// TwinCAT 3 PLC project Library
// Title: lcls-twincat-motion
// Company: SLAC
// ProjectVersion: 0.0.0
// ProgramVersion: 3.1.4026.17
// libraries:
//   LCLS General, * (SLAC)
//   lcls-twincat-math, * (SLAC - LCLS)
//   LCLS_OOPMotion, * (SLAC)
//   PMPS, * (SLAC - LCLS)
//   Tc2_EtherCAT, * (Beckhoff Automation GmbH)
//   Tc2_Math, * (Beckhoff Automation GmbH)
//   Tc2_MC2, * (Beckhoff Automation GmbH)
//   Tc2_Standard, * (Beckhoff Automation GmbH)
//   Tc2_System, * (Beckhoff Automation GmbH)
//   Tc2_Utilities, * (Beckhoff Automation GmbH)
//   Tc3_IPCDiag, * (Beckhoff Automation GmbH)
//   Tc3_JsonXml, * (Beckhoff Automation GmbH)
//   Tc3_Module, * (Beckhoff Automation GmbH)
//   TcUnit, * (www.tcunit.org)
// project tree:
//   DUTs/Deprecated/ ENUM_MotionRequest.TcDUT, DUT_MotionPneumaticActuator.TcDUT, DUT_MotionStage.TcDUT, DUT_PositionState.TcDUT, EL5042_Status.TcDUT, ENUM_EpicsHomeCmd.TcDUT, ENUM_EpicsInOut.TcDUT, ENUM_EpicsInOut_INT.TcDUT, ENUM_EpicsMotorCmd.TcDUT, ENUM_MotionFFType.TcDUT, ENUM_PnuematicActuatorPositionState.TcDUT, ENUM_StageBrakeMode.TcDUT, ENUM_StageEnableMode.TcDUT, ENUM_StatePMPSStatus.TcDUT
//   DUTs/DS402/ E_DS402DriveState.TcDUT, E_DS402EGU.TcDUT, E_MCS2HomeMethod.TcDUT, E_MCS2OpMode.TcDUT, E_MCS2OpModeReq.TcDUT, E_HomeStates.TcDUT (not stored), E_Module.TcDUT, E_MoveDoneCause.TcDUT, E_MoveMode.TcDUT, E_MoveState.TcDUT, E_StartupState.TcDUT, ST_ChannelState.TcDUT, ST_DS402Drive.TcDUT, ST_DS402DriveStatus.TcDUT (not stored), ST_MCS2ChanParameter.TcDUT
//   DUTs/ E_EpicsHomeCmd.TcDUT, ST_AxisParameterSetExposed.TcDUT, E_LCLSMotionError.TcDUT, E_MotionFFType.TcDUT, E_StatePMPSStatus.TcDUT, ST_MotionEpicsInterface.TcDUT, ST_MotionStage.TcDUT, ST_PositionState.TcDUT, ST_StateEpicsToPlc.TcDUT, ST_StatePlcToEpics.TcDUT, ST_StatePMPSEpicsToPlc.TcDUT, ST_EL5042_Status.TcDUT, E_EpicsInOut.TcDUT, E_EpicsMotorCmd.TcDUT, E_MotionRequest.TcDUT, E_StageBrakeMode.TcDUT, E_StageEnableMode.TcDUT, ST_MotionPneumaticActuator.TcDUT, E_PnuematicActuatorPositionState.TcDUT, ST_RenishawAbsEnc.TcDUT, ST_StatePMPSPlcToEpics.TcDUT
//   GVLs/ MOTION_GVL.TcGVL, MotionConstants.TcGVL
//   / PlcTask.TcTTO
//   POUs/Deprecated/ FB_EpicsInOut.TcPOU, FB_PositionStateBase.TcPOU, FB_PositionStateBase_WithPMPS.TcPOU, FB_PositionStateBase_WithPMPS_Test.TcPOU, FB_PositionStateInOut.TcPOU, FB_PositionStateInOut_WithPMPS.TcPOU, FB_PositionStateInOut_WithPMPS_Test.TcPOU, FB_PositionStateManager.TcPOU, FB_PositionStatePMPS.TcPOU, FB_PositionStatePMPS_Base.TcPOU, FB_PositionStatePMPS_Test.TcPOU, FB_StatePTPMove.TcPOU
//   POUs/ImplicitChecks/ CheckBounds.TcPOU, CheckDivDInt.TcPOU, CheckDivLInt.TcPOU, CheckDivLReal.TcPOU, CheckDivReal.TcPOU
//   POUs/Motion/DS402/ FB_MotionStageE727.TcPOU (excluded from build)
//   POUs/Motion/DS402/MCS2/ FB_MCS2Calibrate.TcPOU, FB_MCS2DriveManager.TcPOU, FB_MCS2Home.TcPOU, FB_MCS2ReadParams.TcPOU (excluded from build), FB_MCS2StepMode.TcPOU, FB_MotionStageMCS2.TcPOU, FB_ReadChanParameters.TcPOU, FB_ReadDriveCodes.TcPOU, FB_WriteCalibrationParameters.TcPOU (excluded from build), FB_WriteHomeParameters.TcPOU (excluded from build), FB_WriteChanParameters.TcPOU, F_MCS2ErrorCodeLookup.TcPOU, FB_WriteStepModeParameters.TcPOU (excluded from build)
//   POUs/Motion/ FB_EncoderValue.TcPOU, FB_EncSaveRestore.TcPOU, FB_LogMotionError.TcPOU, FB_MotionBacklashCompensation.TcPOU, FB_MotionHoming.TcPOU, FB_MotionRequest.TcPOU, FB_MotionStage.TcPOU, FB_MotionStageNCParams.TcPOU, FB_MotionStageSim.TcPOU, FB_MotionPneumaticActuator.TcPOU, FB_MotionVirtualFrame.TcPOU
//   POUs/Motion/Gantry/ FB_GantryAutoCoupling.TcPOU, FB_GantryDiffVirtualLimitSwitch.TcPOU
//   POUs/Motion/PMPS/ FB_EncErrorFFO.TcPOU, FB_MiscStatesErrorFFO.TcPOU, FB_MotionBPTM.TcPOU, FB_MotionClearAsserts.TcPOU, FB_MotionReadPMPSDBND.TcPOU, FB_PerMotorFFOND.TcPOU, FB_NCErrorFFO.TcPOU, FB_PositionStatePMPS1D.TcPOU, FB_PositionStatePMPS2D.TcPOU, FB_PositionStatePMPS3D.TcPOU, FB_PositionStatePMPSND_Core.TcPOU, FB_Standard_PMPSDB.TcPOU, FB_StatePMPSEnables.TcPOU, FB_StatePMPSEnablesND.TcPOU
//   POUs/Motion/States/Examples/ FB_PositionState1D_InOut.TcPOU, FB_PositionStatePMPS2D_InOut.TcPOU, FB_PositionStatePMPS1D_InOut.TcPOU, FB_PositionState2D_InOut.TcPOU
//   POUs/Motion/States/ FB_PositionState2D.TcPOU, FB_PositionState3D.TcPOU, FB_PositionStateND_Core.TcPOU, FB_PositionStateMove.TcPOU, FB_PositionState1D.TcPOU, FB_PositionStateMoveND.TcPOU, FB_PositionStateRead.TcPOU, FB_PositionStateReadND.TcPOU, FB_StateSetupHelper.TcPOU, FB_StatesInputHandler.TcPOU
//   POUs/Motion/States/Helpers/ FB_RawCountConverter.TcPOU, F_AtPositionState.TcPOU, F_PosOverLowerBound.TcPOU, F_PosUnderUpperBound.TcPOU, F_PosWithinDelta.TcPOU
//   POUs/Motion/States/Internals/ FB_PositionStateInternal.TcPOU, FB_PositionStateInternalND.TcPOU, FB_PositionStateLock.TcPOU
//   POUs/Motion/Utils/ FB_SetEnables.TcPOU, F_MotionErrorCodeLookup.TcPOU
//   POUs/MotorTesting/ FB_MicroStepCountTest.TcPOU
//   tc_mca_std_lib/DUTs/ DUT_AxisStatus_v0_01.TcDUT (not stored)
//   tc_mca_std_lib/GVLs/ GVL.TcGVL (not stored)
//   tc_mca_std_lib/POUs/ChangeConfig/ FB_ReadFloatParameter.TcPOU (not stored), FB_ReadParameterInNc_v1_00.TcPOU (not stored), FB_WriteFloatParameter.TcPOU (not stored), FB_WriteParameterInNc_v1_00.TcPOU (not stored)
//   tc_mca_std_lib/POUs/ErrorHandling/ DUT_ErrorState.TcDUT (not stored), DUT_TerminalError.TcDUT (not stored), FB_ErrorList.TcPOU (not stored), FB_TerminalError.TcPOU (not stored), GVL_ErrorSystem.TcGVL (not stored), ST_ErrorSystem.TcDUT (not stored)
//   tc_mca_std_lib/POUs/Hardware/EtherCAT_Terminals/Analog_Inputs/ EL3174_0002.TcPOU (not stored), EL3214.TcPOU (not stored), EL3255.TcPOU (not stored), FB_CalculateFrequency_3702_v0_01.TcPOU (not stored)
//   tc_mca_std_lib/POUs/Hardware/EtherCAT_Terminals/Digital_Inputs/ EL1008.TcPOU (not stored), EL1018.TcPOU (not stored), EL1808.TcPOU (not stored), EL1809.TcPOU (not stored), EL1819.TcPOU (not stored), FB_EL1252ASM_v1_00.TcPOU (not stored)
//   tc_mca_std_lib/POUs/Hardware/EtherCAT_Terminals/Digital_Outputs/ EL2014.TcPOU (not stored), EL2252.TcPOU (not stored), EL2808.TcPOU (not stored), EL2819.TcPOU (not stored)
//   tc_mca_std_lib/POUs/Hardware/EtherCAT_Terminals/Digital_Outputs/External_Types/ dutEL2521_Ctrl.TcDUT (not stored), dutEL2521_Status.TcDUT (not stored)
//   tc_mca_std_lib/POUs/Hardware/EtherCAT_Terminals/Measuring_Terminals/ EL5002.TcPOU (not stored), EL5021.TcPOU (not stored), EL5042.TcPOU (not stored), EL5101.TcPOU (not stored)
//   tc_mca_std_lib/POUs/Hardware/EtherCAT_Terminals/Motion/ EL7211_v1_00.TcPOU (not stored), EL9576_v1_00.TcPOU (not stored)
//   tc_mca_std_lib/POUs/Hardware/EtherCAT_Terminals/System/ EL9410.TcPOU (not stored), EL9505.TcPOU (not stored)
//   tc_mca_std_lib/POUs/Hardware/Other/ EK1200.TcPOU (not stored)
//   tc_mca_std_lib/POUs/Motion/ FB_DriveVirtual.TcPOU (not stored), FB_NcAxis.TcPOU (not stored)
//   tc_mca_std_lib/POUs/Motion/Homing/ FB_HomeDirect.TcPOU (not stored), FB_HomeFinish.TcPOU (not stored), FB_HomePrepare.TcPOU (not stored), FB_HomeReadNcVelocities.TcPOU (not stored), FB_HomeReadSoftLimEnable.TcPOU (not stored), FB_HomeToSwitch.TcPOU (not stored), FB_HomeVirtual.TcPOU (not stored), FB_HomeWriteNcVelocities.TcPOU (not stored), FB_HomeWriteSoftLimEnable.TcPOU (not stored)
//   Tests/ FB_AtPositionState_Test.TcPOU, FB_AxisParameterSetExposed_Test.TcPOU, FB_MiscStatesErrorFFO_Test.TcPOU, FB_MotionBPTM_Test.TcPOU, FB_MCS2DriveManager_Test.TcPOU, FB_MotionClearAsserts_Test.TcPOU, FB_MotionReadPMPSDBND_Test.TcPOU, FB_MotionVirtualFrame_Test.TcPOU, FB_NCErrorFFO_Test.TcPOU, FB_PerMotorFFOND_Test.TcPOU, FB_PositionStateMoveND_Test.TcPOU, FB_PositionStateMove_Test.TcPOU, FB_PositionStatePMPSND_Test.TcPOU, FB_PositionStateReadND_Test.TcPOU, FB_PositionStateRead_Test.TcPOU, FB_PositionStateND_Test.TcPOU, FB_PowerEnableMode_Test.TcPOU, FB_MotionBacklashCompensation_Test.TcPOU, FB_StatePMPSEnablesND_Test.TcPOU, FB_StatePMPSEnables_Test.TcPOU, FB_StateSetupHelper_Test.TcPOU, FB_TestHelperSetAndMove_Test.TcPOU, FB_TestStateInitTiming.TcPOU, PRG_TEST.TcPOU
//   Tests/Helpers/ E_TestStates.TcDUT, FB_CauseNCError.TcPOU, FB_MotionStageSetAndMoveHelper.TcPOU, FB_MotionStageSetHelper.TcPOU, FB_MotorTestSuite.TcPOU, FB_PMPSJsonTestHelper.TcPOU, FB_TestHelperSetAndMove.TcPOU
// real-time tasks:
//   TASK PlcTask: cycle T#10ms, priority 20, ADS port 350
// motion (NC):
//   TASK NC-Task 1 SAF: cycle T#1ms, priority 4, ADS port 501
//   TASK NC-Task 1 SVB: cycle T#10ms, priority 8, ADS port 511
//   AXIS Axis_PositionStateRead_Test (id 3)
//     OtherSettings: AllowMotionCmdToSlave=true
//     encoder EncType=1
//     drive DrvType=5
//       Analog: ScaleFactorActTorque=0.1
//     controller CtrType=1
//       CtrPara: PriorControlFactor=1
//         Observer: BandWidth=20
//   AXIS Axis_AtPositionState_Test (id 4)
//     OtherSettings: AllowMotionCmdToSlave=true
//     encoder EncType=1
//     drive DrvType=5
//       Analog: ScaleFactorActTorque=0.1
//     controller CtrType=1
//       CtrPara: PriorControlFactor=1
//         Observer: BandWidth=20
//   AXIS Axis_TestHelperSetAndMove_Test (id 5)
//     OtherSettings: AllowMotionCmdToSlave=true
//     encoder EncType=1
//     drive DrvType=5
//       Analog: ScaleFactorActTorque=0.1
//     controller CtrType=1
//       CtrPara: PriorControlFactor=1
//         Observer: BandWidth=20
//   AXIS Axis_PositionStateReadND_Test_1 (id 6)
//     OtherSettings: AllowMotionCmdToSlave=true
//     encoder EncType=1
//     drive DrvType=5
//       Analog: ScaleFactorActTorque=0.1
//       TimeComp: TaskDelayCycles=1
//     controller CtrType=1
//       CtrPara: PriorControlFactor=1
//         Observer: BandWidth=20
//   AXIS Axis_PositionStateReadND_Test_2 (id 7)
//     OtherSettings: AllowMotionCmdToSlave=true
//     encoder EncType=1
//     drive DrvType=5
//       Analog: ScaleFactorActTorque=0.1
//       TimeComp: TaskDelayCycles=1
//     controller CtrType=1
//       CtrPara: PriorControlFactor=1
//         Observer: BandWidth=20
//   AXIS Axis_PositionStateReadND_Test_3 (id 8)
//     OtherSettings: AllowMotionCmdToSlave=true
//     encoder EncType=1
//     drive DrvType=5
//       Analog: ScaleFactorActTorque=0.1
//       TimeComp: TaskDelayCycles=1
//     controller CtrType=1
//       CtrPara: PriorControlFactor=1
//         Observer: BandWidth=20
//   AXIS Axis_PositionStateMove_Test (id 9)
//     OtherSettings: AllowMotionCmdToSlave=true
//     encoder EncType=1
//     drive DrvType=5
//       Analog: ScaleFactorActTorque=0.1
//     controller CtrType=1
//       CtrPara: PriorControlFactor=1
//         Observer: BandWidth=20
//   AXIS Axis_PositionStateMoveND_Test_1 (id 10)
//     OtherSettings: AllowMotionCmdToSlave=true
//     encoder EncType=1
//     drive DrvType=5
//       Analog: ScaleFactorActTorque=0.1
//     controller CtrType=1
//       CtrPara: PriorControlFactor=1
//         Observer: BandWidth=20
//   AXIS Axis_PositionStateMoveND_Test_2 (id 11)
//     OtherSettings: AllowMotionCmdToSlave=true
//     encoder EncType=1
//     drive DrvType=5
//       Analog: ScaleFactorActTorque=0.1
//     controller CtrType=1
//       CtrPara: PriorControlFactor=1
//         Observer: BandWidth=20
//   AXIS Axis_PositionStateMoveND_Test_3 (id 12)
//     OtherSettings: AllowMotionCmdToSlave=true
//     encoder EncType=1
//     drive DrvType=5
//       Analog: ScaleFactorActTorque=0.1
//     controller CtrType=1
//       CtrPara: PriorControlFactor=1
//         Observer: BandWidth=20
//   AXIS Axis_PositionStateND_Test_1 (id 13)
//     OtherSettings: AllowMotionCmdToSlave=true
//     encoder EncType=1
//     drive DrvType=5
//       Analog: ScaleFactorActTorque=0.1
//       TimeComp: TaskDelayCycles=1
//     controller CtrType=1
//       CtrPara: PriorControlFactor=1
//         Observer: BandWidth=20
//   AXIS Axis_PositionStateND_Test_2 (id 14)
//     OtherSettings: AllowMotionCmdToSlave=true
//     encoder EncType=1
//     drive DrvType=5
//       Analog: ScaleFactorActTorque=0.1
//       TimeComp: TaskDelayCycles=1
//     controller CtrType=1
//       CtrPara: PriorControlFactor=1
//         Observer: BandWidth=20
//   AXIS Axis_PositionStateND_Test_3 (id 15)
//     OtherSettings: AllowMotionCmdToSlave=true
//     encoder EncType=1
//     drive DrvType=5
//       Analog: ScaleFactorActTorque=0.1
//       TimeComp: TaskDelayCycles=1
//     controller CtrType=1
//       CtrPara: PriorControlFactor=1
//         Observer: BandWidth=20
//   AXIS Axis_NCErrorFFO_Test (id 16)
//     OtherSettings: AllowMotionCmdToSlave=true
//     encoder EncType=1
//     drive DrvType=5
//       Analog: ScaleFactorActTorque=0.1
//     controller CtrType=1
//       CtrPara: PriorControlFactor=1
//         Observer: BandWidth=20
//   AXIS Axis_PositionStatePMPSND_Test_1 (id 17)
//     OtherSettings: AllowMotionCmdToSlave=true
//     encoder EncType=1
//     drive DrvType=5
//       Analog: ScaleFactorActTorque=0.1
//     controller CtrType=1
//       CtrPara: PriorControlFactor=1
//         Observer: BandWidth=20
//   AXIS Axis_PositionStatePMPSND_Test_2 (id 18)
//     OtherSettings: AllowMotionCmdToSlave=true
//     encoder EncType=1
//     drive DrvType=5
//       Analog: ScaleFactorActTorque=0.1
//     controller CtrType=1
//       CtrPara: PriorControlFactor=1
//         Observer: BandWidth=20
//   AXIS Axis_PositionStatePMPSND_Test_3 (id 19)
//     OtherSettings: AllowMotionCmdToSlave=true
//     encoder EncType=1
//     drive DrvType=5
//       Analog: ScaleFactorActTorque=0.1
//     controller CtrType=1
//       CtrPara: PriorControlFactor=1
//         Observer: BandWidth=20
//   AXIS Axis_StatePMPSEnable_Test (id 20)
//     OtherSettings: AllowMotionCmdToSlave=true
//     encoder EncType=1
//     drive DrvType=5
//       Analog: ScaleFactorActTorque=0.1
//       TimeComp: TaskDelayCycles=1
//     controller CtrType=1
//       CtrPara: PriorControlFactor=1
//         Observer: BandWidth=20
//   AXIS Axis_PositionStateReadND_Test_4 (id 21)
//     OtherSettings: AllowMotionCmdToSlave=true
//     encoder EncType=1
//     drive DrvType=5
//       Analog: ScaleFactorActTorque=0.1
//     controller CtrType=1
//       CtrPara: PriorControlFactor=1
//         Observer: BandWidth=20
//   AXIS Axis_PositionStateReadND_Test_5 (id 22)
//     OtherSettings: AllowMotionCmdToSlave=true
//     encoder EncType=1
//     drive DrvType=5
//       Analog: ScaleFactorActTorque=0.1
//     controller CtrType=1
//       CtrPara: PriorControlFactor=1
//         Observer: BandWidth=20
//   AXIS Axis_TestStateInitTiming (id 1)
//     OtherSettings: AllowMotionCmdToSlave=true
//     encoder EncType=1
//     drive DrvType=5
//       Analog: TorqueSetpointScale=10, ScaleFactorActTorque=0.1
//     controller CtrType=1
//       CtrPara: PriorControlFactor=1
//         Observer: BandWidth=20
//   AXIS Axis_AxisParameter_Test (id 2)
//     Dynamic: AccelerationMaximum=2, DecelerationMaximum=3
//     Velo: Maximum=1
//     PositionAreaControl: Range=1
//     OtherSettings: AllowMotionCmdToSlave=true
//     encoder EncType=1
//       EncPara: Offset=12
//         SoftEndMinControl: Enable=true, Range=4
//         SoftEndMaxControl: Enable=true, Range=5
//     drive DrvType=5
//       Analog: TorqueSetpointScale=10, ScaleFactorActTorque=0.1
//       TimeComp: TaskDelayCycles=1
//     controller CtrType=1
//       CtrPara: PriorControlFactor=1
//         PosDiffControl: Range=6, Time=7
//         Observer: BandWidth=20
//   AXIS Axis_PowerEnableMode_Test (id 29) // Test axis for stmotionStage Axis Power Enable Mode control
//     OtherSettings: AllowMotionCmdToSlave=true
//     encoder EncType=1
//     drive DrvType=5
//       Analog: TorqueSetpointScale=10, ScaleFactorActTorque=0.1
//       TimeComp: TaskDelayCycles=1
//     controller CtrType=1
//       CtrPara: PriorControlFactor=1
//         Observer: BandWidth=20
//   AXIS Axis_BacklashCompensation_Test (id 30)
//     OtherSettings: AllowMotionCmdToSlave=true
//     encoder EncType=1
//       ActPosCorrection: Enable=true
//     drive DrvType=5
//       Analog: TorqueSetpointScale=10, ScaleFactorActTorque=0.1
//     controller CtrType=1
//       CtrPara: PriorControlFactor=1
//         Observer: BandWidth=20
//   AXIS Axis_NewArchMcMotionBlocks_Test (id 31)
//     OtherSettings: AllowMotionCmdToSlave=true
//     encoder EncType=1
//     drive DrvType=5
//       Analog: TorqueSetpointScale=10, ScaleFactorActTorque=0.1
//       TimeComp: TaskDelayCycles=1
//     controller CtrType=1
//       CtrPara: PriorControlFactor=1
//         Observer: BandWidth=20
//   AXIS Axis_MotionVirtualFrameRx_Test (id 23)
//     OtherSettings: AllowMotionCmdToSlave=true
//     encoder EncType=1
//     drive DrvType=5
//       Analog: TorqueSetpointScale=10, ScaleFactorActTorque=0.1
//     controller CtrType=1
//       CtrPara: PriorControlFactor=1
//         Observer: BandWidth=20
//   AXIS Axis_MotionVirtualFrameRy_Test (id 24)
//     OtherSettings: AllowMotionCmdToSlave=true
//     encoder EncType=1
//     drive DrvType=5
//       Analog: TorqueSetpointScale=10, ScaleFactorActTorque=0.1
//     controller CtrType=1
//       CtrPara: PriorControlFactor=1
//         Observer: BandWidth=20
//   AXIS Axis_MotionVirtualFrameRz_Test (id 25)
//     OtherSettings: AllowMotionCmdToSlave=true
//     encoder EncType=1
//     drive DrvType=5
//       Analog: TorqueSetpointScale=10, ScaleFactorActTorque=0.1
//     controller CtrType=1
//       CtrPara: PriorControlFactor=1
//         Observer: BandWidth=20
//   AXIS Axis_MotionVirtualFrameVx_Test (id 26)
//     OtherSettings: AllowMotionCmdToSlave=true
//     encoder EncType=7
//       EncPara: ScaleFactorNumerator=1e-06, MaxCount=#xffffffff, ReferenceSystem=1
//     drive DrvType=5
//       Analog: TorqueSetpointScale=10, ScaleFactorActTorque=0.1
//       TimeComp: TaskDelayCycles=1
//     controller CtrType=1
//       CtrPara: PriorControlFactor=1
//         PosDiffControl: Enable=false
//         Observer: BandWidth=20
//   AXIS Axis_MotionVirtualFrameVy_Test (id 27)
//     OtherSettings: AllowMotionCmdToSlave=true
//     encoder EncType=7
//       EncPara: ScaleFactorNumerator=1e-06, MaxCount=#xffffffff, ReferenceSystem=1
//     drive DrvType=5
//       Analog: TorqueSetpointScale=10, ScaleFactorActTorque=0.1
//       TimeComp: TaskDelayCycles=1
//     controller CtrType=1
//       CtrPara: PriorControlFactor=1
//         PosDiffControl: Enable=false
//         Observer: BandWidth=20
//   AXIS Axis_MotionVirtualFrameVz_Test (id 28)
//     OtherSettings: AllowMotionCmdToSlave=true
//     encoder EncType=7
//       EncPara: ScaleFactorNumerator=1e-06, MaxCount=#xffffffff, ReferenceSystem=1
//     drive DrvType=5
//       Analog: TorqueSetpointScale=10, ScaleFactorActTorque=0.1
//       TimeComp: TaskDelayCycles=1
//     controller CtrType=1
//       CtrPara: PriorControlFactor=1
//         PosDiffControl: Enable=false
//         Observer: BandWidth=20
// variable links:
//   Library Instance <-> NC-Task 1 SAF/Axes/Axis_AtPositionState_Test
//     PlcTask Inputs/PRG_TEST.fb_AtPositionState_Test.stMotionStage.Axis.NcToPlc <-> Outputs/ToPlc
//     PlcTask Outputs/PRG_TEST.fb_AtPositionState_Test.stMotionStage.Axis.PlcToNc <-> Inputs/FromPlc
//   Library Instance <-> NC-Task 1 SAF/Axes/Axis_AxisParameter_Test
//     PlcTask Inputs/PRG_TEST.fb_AxisParameterSetExposed_Test.stMotionStage.Axis.NcToPlc <-> Outputs/ToPlc
//     PlcTask Outputs/PRG_TEST.fb_AxisParameterSetExposed_Test.stMotionStage.Axis.PlcToNc <-> Inputs/FromPlc
//   Library Instance <-> NC-Task 1 SAF/Axes/Axis_BacklashCompensation_Test
//     PlcTask Inputs/PRG_TEST.fb_MotionBacklashCompensation_Test.stMotionStage.Axis.NcToPlc <-> Outputs/ToPlc
//     PlcTask Outputs/PRG_TEST.fb_MotionBacklashCompensation_Test.stMotionStage.Axis.PlcToNc <-> Inputs/FromPlc
//   Library Instance <-> NC-Task 1 SAF/Axes/Axis_MotionVirtualFrameRx_Test
//     PlcTask Inputs/PRG_TEST.fbMotionVirtualFrameTest.stMotionStageRx.Axis.NcToPlc <-> Outputs/ToPlc
//     PlcTask Outputs/PRG_TEST.fbMotionVirtualFrameTest.stMotionStageRx.Axis.PlcToNc <-> Inputs/FromPlc
//   Library Instance <-> NC-Task 1 SAF/Axes/Axis_MotionVirtualFrameRy_Test
//     PlcTask Inputs/PRG_TEST.fbMotionVirtualFrameTest.stMotionStageRy.Axis.NcToPlc <-> Outputs/ToPlc
//     PlcTask Outputs/PRG_TEST.fbMotionVirtualFrameTest.stMotionStageRy.Axis.PlcToNc <-> Inputs/FromPlc
//   Library Instance <-> NC-Task 1 SAF/Axes/Axis_MotionVirtualFrameRz_Test
//     PlcTask Inputs/PRG_TEST.fbMotionVirtualFrameTest.stMotionStageRz.Axis.NcToPlc <-> Outputs/ToPlc
//     PlcTask Outputs/PRG_TEST.fbMotionVirtualFrameTest.stMotionStageRz.Axis.PlcToNc <-> Inputs/FromPlc
//   Library Instance <-> NC-Task 1 SAF/Axes/Axis_MotionVirtualFrameVx_Test
//     PlcTask Inputs/PRG_TEST.fbMotionVirtualFrameTest.stMotionStageVx.Axis.NcToPlc <-> Outputs/ToPlc
//     PlcTask Outputs/PRG_TEST.fbMotionVirtualFrameTest.nPositionCountsVx <-> Enc/Inputs/In/nDataIn1
//     PlcTask Outputs/PRG_TEST.fbMotionVirtualFrameTest.stMotionStageVx.Axis.PlcToNc <-> Inputs/FromPlc
//   Library Instance <-> NC-Task 1 SAF/Axes/Axis_MotionVirtualFrameVy_Test
//     PlcTask Inputs/PRG_TEST.fbMotionVirtualFrameTest.stMotionStageVy.Axis.NcToPlc <-> Outputs/ToPlc
//     PlcTask Outputs/PRG_TEST.fbMotionVirtualFrameTest.nPositionCountsVy <-> Enc/Inputs/In/nDataIn1
//     PlcTask Outputs/PRG_TEST.fbMotionVirtualFrameTest.stMotionStageVy.Axis.PlcToNc <-> Inputs/FromPlc
//   Library Instance <-> NC-Task 1 SAF/Axes/Axis_MotionVirtualFrameVz_Test
//     PlcTask Inputs/PRG_TEST.fbMotionVirtualFrameTest.stMotionStageVz.Axis.NcToPlc <-> Outputs/ToPlc
//     PlcTask Outputs/PRG_TEST.fbMotionVirtualFrameTest.nPositionCountsVz <-> Enc/Inputs/In/nDataIn1
//     PlcTask Outputs/PRG_TEST.fbMotionVirtualFrameTest.stMotionStageVz.Axis.PlcToNc <-> Inputs/FromPlc
//   Library Instance <-> NC-Task 1 SAF/Axes/Axis_NCErrorFFO_Test
//     PlcTask Inputs/PRG_TEST.fb_NCErrorFFO_Test.stMotionStage.Axis.NcToPlc <-> Outputs/ToPlc
//     PlcTask Outputs/PRG_TEST.fb_NCErrorFFO_Test.stMotionStage.Axis.PlcToNc <-> Inputs/FromPlc
//   Library Instance <-> NC-Task 1 SAF/Axes/Axis_PositionStateMoveND_Test_1
//     PlcTask Inputs/PRG_TEST.fb_PositionStateMoveND_Test.astMotionStage[1].Axis.NcToPlc <-> Outputs/ToPlc
//     PlcTask Outputs/PRG_TEST.fb_PositionStateMoveND_Test.astMotionStage[1].Axis.PlcToNc <-> Inputs/FromPlc
//   Library Instance <-> NC-Task 1 SAF/Axes/Axis_PositionStateMoveND_Test_2
//     PlcTask Inputs/PRG_TEST.fb_PositionStateMoveND_Test.astMotionStage[2].Axis.NcToPlc <-> Outputs/ToPlc
//     PlcTask Outputs/PRG_TEST.fb_PositionStateMoveND_Test.astMotionStage[2].Axis.PlcToNc <-> Inputs/FromPlc
//   Library Instance <-> NC-Task 1 SAF/Axes/Axis_PositionStateMoveND_Test_3
//     PlcTask Inputs/PRG_TEST.fb_PositionStateMoveND_Test.astMotionStage[3].Axis.NcToPlc <-> Outputs/ToPlc
//     PlcTask Outputs/PRG_TEST.fb_PositionStateMoveND_Test.astMotionStage[3].Axis.PlcToNc <-> Inputs/FromPlc
//   Library Instance <-> NC-Task 1 SAF/Axes/Axis_PositionStateMove_Test
//     PlcTask Inputs/PRG_TEST.fb_PositionStateMove_Test.stMotionStage.Axis.NcToPlc <-> Outputs/ToPlc
//     PlcTask Outputs/PRG_TEST.fb_PositionStateMove_Test.stMotionStage.Axis.PlcToNc <-> Inputs/FromPlc
//   Library Instance <-> NC-Task 1 SAF/Axes/Axis_PositionStateND_Test_1
//     PlcTask Inputs/PRG_TEST.fb_PositionStateND_Test.stMotionStage1.Axis.NcToPlc <-> Outputs/ToPlc
//     PlcTask Outputs/PRG_TEST.fb_PositionStateND_Test.stMotionStage1.Axis.PlcToNc <-> Inputs/FromPlc
//   Library Instance <-> NC-Task 1 SAF/Axes/Axis_PositionStateND_Test_2
//     PlcTask Inputs/PRG_TEST.fb_PositionStateND_Test.stMotionStage2.Axis.NcToPlc <-> Outputs/ToPlc
//     PlcTask Outputs/PRG_TEST.fb_PositionStateND_Test.stMotionStage2.Axis.PlcToNc <-> Inputs/FromPlc
//   Library Instance <-> NC-Task 1 SAF/Axes/Axis_PositionStateND_Test_3
//     PlcTask Inputs/PRG_TEST.fb_PositionStateND_Test.stMotionStage3.Axis.NcToPlc <-> Outputs/ToPlc
//     PlcTask Outputs/PRG_TEST.fb_PositionStateND_Test.stMotionStage3.Axis.PlcToNc <-> Inputs/FromPlc
//   Library Instance <-> NC-Task 1 SAF/Axes/Axis_PositionStatePMPSND_Test_1
//     PlcTask Inputs/PRG_TEST.fb_PositionStatePMPSND_Test.stMotionStage1.Axis.NcToPlc <-> Outputs/ToPlc
//     PlcTask Outputs/PRG_TEST.fb_PositionStatePMPSND_Test.stMotionStage1.Axis.PlcToNc <-> Inputs/FromPlc
//   Library Instance <-> NC-Task 1 SAF/Axes/Axis_PositionStatePMPSND_Test_2
//     PlcTask Inputs/PRG_TEST.fb_PositionStatePMPSND_Test.stMotionStage2.Axis.NcToPlc <-> Outputs/ToPlc
//     PlcTask Outputs/PRG_TEST.fb_PositionStatePMPSND_Test.stMotionStage2.Axis.PlcToNc <-> Inputs/FromPlc
//   Library Instance <-> NC-Task 1 SAF/Axes/Axis_PositionStatePMPSND_Test_3
//     PlcTask Inputs/PRG_TEST.fb_PositionStatePMPSND_Test.stMotionStage3.Axis.NcToPlc <-> Outputs/ToPlc
//     PlcTask Outputs/PRG_TEST.fb_PositionStatePMPSND_Test.stMotionStage3.Axis.PlcToNc <-> Inputs/FromPlc
//   Library Instance <-> NC-Task 1 SAF/Axes/Axis_PositionStateReadND_Test_1
//     PlcTask Inputs/PRG_TEST.fb_PositionStateReadND_Test.astMotionStage[1].Axis.NcToPlc <-> Outputs/ToPlc
//     PlcTask Outputs/PRG_TEST.fb_PositionStateReadND_Test.astMotionStage[1].Axis.PlcToNc <-> Inputs/FromPlc
//   Library Instance <-> NC-Task 1 SAF/Axes/Axis_PositionStateReadND_Test_2
//     PlcTask Inputs/PRG_TEST.fb_PositionStateReadND_Test.astMotionStage[2].Axis.NcToPlc <-> Outputs/ToPlc
//     PlcTask Outputs/PRG_TEST.fb_PositionStateReadND_Test.astMotionStage[2].Axis.PlcToNc <-> Inputs/FromPlc
//   Library Instance <-> NC-Task 1 SAF/Axes/Axis_PositionStateReadND_Test_3
//     PlcTask Inputs/PRG_TEST.fb_PositionStateReadND_Test.astMotionStage[3].Axis.NcToPlc <-> Outputs/ToPlc
//     PlcTask Outputs/PRG_TEST.fb_PositionStateReadND_Test.astMotionStage[3].Axis.PlcToNc <-> Inputs/FromPlc
//   Library Instance <-> NC-Task 1 SAF/Axes/Axis_PositionStateReadND_Test_4
//     PlcTask Inputs/PRG_TEST.fb_PositionStateReadND_Test.astSqMotionStage[1].Axis.NcToPlc <-> Outputs/ToPlc
//     PlcTask Outputs/PRG_TEST.fb_PositionStateReadND_Test.astSqMotionStage[1].Axis.PlcToNc <-> Inputs/FromPlc
//   Library Instance <-> NC-Task 1 SAF/Axes/Axis_PositionStateReadND_Test_5
//     PlcTask Inputs/PRG_TEST.fb_PositionStateReadND_Test.astSqMotionStage[2].Axis.NcToPlc <-> Outputs/ToPlc
//     PlcTask Outputs/PRG_TEST.fb_PositionStateReadND_Test.astSqMotionStage[2].Axis.PlcToNc <-> Inputs/FromPlc
//   Library Instance <-> NC-Task 1 SAF/Axes/Axis_PositionStateRead_Test
//     PlcTask Inputs/PRG_TEST.fb_PositionStateRead_Test.stMotionStage.Axis.NcToPlc <-> Outputs/ToPlc
//     PlcTask Outputs/PRG_TEST.fb_PositionStateRead_Test.stMotionStage.Axis.PlcToNc <-> Inputs/FromPlc
//   Library Instance <-> NC-Task 1 SAF/Axes/Axis_PowerEnableMode_Test
//     PlcTask Inputs/PRG_TEST.fb_PowerEnableMode_Test.stMotionStage.Axis.NcToPlc <-> Outputs/ToPlc
//     PlcTask Outputs/PRG_TEST.fb_PowerEnableMode_Test.stMotionStage.Axis.PlcToNc <-> Inputs/FromPlc
//   Library Instance <-> NC-Task 1 SAF/Axes/Axis_StatePMPSEnable_Test
//     PlcTask Inputs/PRG_TEST.fb_StatePMPSEnables_Test.stMotionStage.Axis.NcToPlc <-> Outputs/ToPlc
//     PlcTask Outputs/PRG_TEST.fb_StatePMPSEnables_Test.stMotionStage.Axis.PlcToNc <-> Inputs/FromPlc
//   Library Instance <-> NC-Task 1 SAF/Axes/Axis_TestHelperSetAndMove_Test
//     PlcTask Inputs/PRG_TEST.fb_TestHelperSetAndMove_Test.stMotionStage.Axis.NcToPlc <-> Outputs/ToPlc
//     PlcTask Outputs/PRG_TEST.fb_TestHelperSetAndMove_Test.stMotionStage.Axis.PlcToNc <-> Inputs/FromPlc
//   Library Instance <-> NC-Task 1 SAF/Axes/Axis_TestStateInitTiming
//     PlcTask Inputs/PRG_TEST.fb_TestStateInitTiming.stMotionStage.Axis.NcToPlc <-> Outputs/ToPlc
//     PlcTask Outputs/PRG_TEST.fb_TestStateInitTiming.stMotionStage.Axis.PlcToNc <-> Inputs/FromPlc

CONFIGURATION Library
    RESOURCE PLC ON TwinCAT3
        TASK PlcTask(INTERVAL := T#10ms, PRIORITY := 20);
        PROGRAM PRG_TEST WITH PlcTask : PRG_TEST;
    END_RESOURCE
END_CONFIGURATION

// ---- DUTs/Deprecated/ENUM_MotionRequest.TcDUT
{attribute 'obsolete' := 'Use E_MotionRequest'}
TYPE ENUM_MotionRequest : E_MotionRequest; END_TYPE

// ---- DUTs/Deprecated/DUT_MotionPneumaticActuator.TcDUT
{attribute 'obsolete' := 'DUT_MotionPneumaticActuator has been renamed to ST_MotionPneumaticActuator'}
TYPE DUT_MotionPneumaticActuator : ST_MotionPneumaticActuator; END_TYPE

// ---- DUTs/Deprecated/DUT_MotionStage.TcDUT
{attribute 'obsolete' := 'DUT_MotionStage has been renamed to ST_MotionStage'}
TYPE DUT_MotionStage : ST_MotionStage; END_TYPE

// ---- DUTs/Deprecated/DUT_PositionState.TcDUT
{attribute 'obsolete' := 'DUT_PositionState has been renamed to ST_PositionState'}
TYPE DUT_PositionState : ST_PositionState; END_TYPE

// ---- DUTs/Deprecated/EL5042_Status.TcDUT
{attribute 'obsolete' := 'EL5042_Status has been renamed to ST_EL5042_Status'}
TYPE EL5042_Status : ST_EL5042_Status; END_TYPE

// ---- DUTs/Deprecated/ENUM_EpicsHomeCmd.TcDUT
{attribute 'obsolete' := 'Use E_EpicsHomeCmd'}
TYPE ENUM_EpicsHomeCmd : E_EpicsHomeCmd; END_TYPE

// ---- DUTs/Deprecated/ENUM_EpicsInOut.TcDUT
{attribute 'obsolete' := 'Use E_EpicsInOut'}
TYPE ENUM_EpicsInOut : E_EpicsInOut; END_TYPE

// ---- DUTs/Deprecated/ENUM_EpicsInOut_INT.TcDUT
{attribute 'obsolete' := 'Use ENUM_EpicsInOut'}
{attribute 'qualified_only'}
// Example EPICS states enum for use in all versions of the states FBs
// Remove strict attribute for easier handling
TYPE ENUM_EpicsInOut_INT :
(
    UNKNOWN := 0, // UNKNOWN must be in slot 0 or the FB breaks
    OUT := 1, // OUT at slot 1 is a convention
    IN := 2
) INT;
END_TYPE

// ---- DUTs/Deprecated/ENUM_EpicsMotorCmd.TcDUT
{attribute 'obsolete' := 'Use E_EpicsMotorCmd'}
TYPE ENUM_EpicsMotorCmd : E_EpicsMotorCmd; END_TYPE

// ---- DUTs/Deprecated/ENUM_MotionFFType.TcDUT
{attribute 'obsolete' := 'Use E_MotionFFType'}
TYPE ENUM_MotionFFType : E_MotionFFType; END_TYPE

// ---- DUTs/Deprecated/ENUM_PnuematicActuatorPositionState.TcDUT
{attribute 'obsolete' := 'Use E_PnuematicActuatorPositionState'}
TYPE ENUM_PnuematicActuatorPositionState : E_PnuematicActuatorPositionState; END_TYPE

// ---- DUTs/Deprecated/ENUM_StageBrakeMode.TcDUT
{attribute 'obsolete' := 'Use E_StageBrakeMode'}
TYPE ENUM_StageBrakeMode : E_StageBrakeMode; END_TYPE

// ---- DUTs/Deprecated/ENUM_StageEnableMode.TcDUT
{attribute 'obsolete' := 'Use E_StageEnableMode'}
TYPE ENUM_StageEnableMode : E_StageEnableMode; END_TYPE

// ---- DUTs/Deprecated/ENUM_StatePMPSStatus.TcDUT
{attribute 'obsolete' := 'Use E_StatePMPSStatus'}
TYPE ENUM_StatePMPSStatus : E_StatePMPSStatus; END_TYPE

// ---- DUTs/DS402/E_DS402DriveState.TcDUT
{attribute 'qualified_only'}
{attribute 'strict'}
{attribute 'to_string'}
TYPE E_DS402DriveState :
(
    INIT:=0,
    NO_FAULT:=1,
    SWITCH_ON_READY:=2,
    SWITCH_ON:=3,
    OPERATION_ENABLED:=4,
    FAULT:=5,
    FAULT_ACTIVE:=6,
    QUICK_STOP_ACTIVE:=7,
    SWITCH_ON_DISABLED:=8,
    MODE_ERROR:=9,
    WAIT	:= 10,
    DONE:=11
) UINT;
END_TYPE

// ---- DUTs/DS402/E_DS402EGU.TcDUT
{attribute 'qualified_only'}
{attribute 'strict'}
{attribute 'to_string'}
TYPE E_DS402EGU  :
(
    MM:=0,
    UM:=1,
    NM:=2
);
END_TYPE

// ---- DUTs/DS402/E_MCS2HomeMethod.TcDUT
{attribute 'qualified_only'}
{attribute 'strict'}
{attribute 'to_string'}
TYPE E_MCS2HomeMethod :
(
    AutoMethod := -1,
    CurrentPositionMethod := 37
)SINT;
END_TYPE

// ---- DUTs/DS402/E_MCS2OpMode.TcDUT
{attribute 'qualified_only'}
{attribute 'strict'}
{attribute 'to_string'}
TYPE E_MCS2OpMode :
(
    NONE := 0,
    // P-T-P target profil
    PROFILE_POSITION:=1,
    PROFIL_VELOCITY :=3,
    HOME:=6,
    // Cyclic synchronous modes
    CSP :=8,
    CSV :=9,
    CST := 10,
    CSTCA := 11,
    // smartAct MCS2 open loop
    CALIBRATE :=-1,
    STEP :=-4
) SINT;
END_TYPE

// ---- DUTs/DS402/E_MCS2OpModeReq.TcDUT
(*
    User-facing request for the MCS2 drive operating mode, exposed as an EPICS PV.
    This is the source of truth for which DS402 mode the drive runs in; the
    FB_MCS2DriveManager maps each value onto the corresponding E_DS402OpMode and
    switches the drive immediately when this value changes.
    CLOSED_LOOP (default) is closed-loop (CSP / NC) absolute motion.
*)
{attribute 'qualified_only'}
{attribute 'strict'}
{attribute 'to_string'}
TYPE E_MCS2OpModeReq :
(
    CLOSED_LOOP := 0,
    STEP := 1,
    HOME := 2,
    CALIBRATION := 3
) SINT;
END_TYPE

// ---- DUTs/DS402/E_Module.TcDUT
{attribute 'qualified_only'}
{attribute 'to_string'}
// Default CHAN 1, add 0x800 next channel
TYPE E_Module :
(
    CHAN1	:= 1,
    CHAN2	:= 2,
    CHAN3	:= 3
) WORD;
END_TYPE

// ---- DUTs/DS402/E_MoveDoneCause.TcDUT
{attribute 'qualified_only'}
{attribute 'strict'}
{attribute 'to_string'}
TYPE E_MoveDoneCause :
(
    UNKNOWN := 0,           // DEFAULT/UNCATEGORIZED
    MOVEDONE,               // ABSOLUTE MOVE COMPLETED
    STEPMOVEDONE,           // STEP/JOG MOVE COMPLETED
    HOMEDONE,               // HOMING COMPLETED
    CALIBRATIONDONE,        // CALIBRATION COMPLETED
    RESETDONE,              // RESET COMMAND COMPLETED
    HALTDONE,               // MANUAL HALT COMPLETED
    ABORTEDHOME,            // HOME ABORTED
    ABORTEDSTEPMOVE,        // STEP MOVE ABORTED
    ABORTEDCALIBRATION,     // CALIBRATION ABORTED
    REFERENCED,             // AXIS BECAME REFERENCED
    CALIBRATED              // AXIS BECAME CALIBRATED
);
END_TYPE

// ---- DUTs/DS402/E_MoveMode.TcDUT
{attribute 'qualified_only'}
{attribute 'strict'}
{attribute 'to_string'}
TYPE E_MoveMode  :
(
    DISCRETE_JOG:=0,
    DISCRETE_VELOCITY:=1,
    DISCRETE_RELATIVE:=2,
    DISCRETE_ABSOLUTE:=3,
    DISCRETE_MODULO:=4,
    DISCRETE_HOMING:=10
)INT;
END_TYPE

// ---- DUTs/DS402/E_MoveState.TcDUT
{attribute 'qualified_only'}
{attribute 'strict'}
{attribute 'to_string'}
TYPE E_MoveState :
(
    IDLING:=0,
    INIT:=10,
    STARTED:=20,
    IN_PROGRESS :=30,
    REACHED:=40,
    INTERRUPTED:=50,
    DONE:=60,
    ERROR:=-99
);
END_TYPE

// ---- DUTs/DS402/E_StartupState.TcDUT
{attribute 'qualified_only'}
{attribute 'strict'}
{attribute 'to_string'}
TYPE E_StartupState :
(
    STARTUP_IDLE:=0,
    STARTUP_CLEAR,
    STARTUP_RESET_FAULT,
    STARTUP_SHUTDOWN,
    STARTUP_SWITCH_ON,
    STARTUP_ENABLE_OP
);
END_TYPE

// ---- DUTs/DS402/ST_ChannelState.TcDUT
TYPE ST_ChannelState :
STRUCT
    {attribute 'pytmc' := '
        pv: STATE
        io: i
        field: DESC Channel state raw
    '}
    nChannelStateRaw  : DWORD;

    {attribute 'pytmc' := '
        pv: MOVING
        io: i
        field: DESC Actively moving
    '}
    bActivelyMoving         : BOOL;
    {attribute 'pytmc' := '
        pv: CLOSED_LOOP
        io: i
        field: DESC Closed loop active
    '}
    bClosedLoopActive       : BOOL;
    {attribute 'pytmc' := '
        pv: CALIBRATING
        io: i
        field: DESC Calibrating
    '}
    bCalibrating            : BOOL;
    {attribute 'pytmc' := '
        pv: REFERENCING
        io: i
        field: DESC Referencing
    '}
    bReferencing            : BOOL;
    {attribute 'pytmc' := '
        pv: MOVE_DELAYED
        io: i
        field: DESC Move delayed
    '}
    bMoveDelayed            : BOOL;
    {attribute 'pytmc' := '
        pv: SENSOR_PRESENT
        io: i
        field: DESC Sensor present
    '}
    bSensorPresent          : BOOL;
    {attribute 'pytmc' := '
        pv: CALIBRATED
        io: i
        field: DESC Is calibrated
    '}
    bIsCalibrated           : BOOL;
    {attribute 'pytmc' := '
        pv: REFERENCED
        io: i
        field: DESC Is referenced
    '}
    bIsReferenced           : BOOL;
    {attribute 'pytmc' := '
        pv: END_STOP
        io: i
        field: DESC End stop reached
    '}
    bEndStopReached         : BOOL;
    {attribute 'pytmc' := '
        pv: RANGE_LIMIT
        io: i
        field: DESC Range limit reached
    '}
    bRangeLimitReached      : BOOL;
    {attribute 'pytmc' := '
        pv: FOLLOWING_LIMIT
        io: i
        field: DESC Following limit reached
    '}
    bFollowingLimitReached  : BOOL;
    {attribute 'pytmc' := '
        pv: MOVE_FAILED
        io: i
        field: DESC Movement failed
    '}
    bMovementFailed         : BOOL;
    {attribute 'pytmc' := '
        pv: STREAMING
        io: i
        field: DESC Is streaming
    '}
    bIsStreaming            : BOOL;
    {attribute 'pytmc' := '
        pv: OVERLOAD
        io: i
        field: DESC Positioner overload
    '}
    bPositionerOverload     : BOOL;
    {attribute 'pytmc' := '
        pv: OVER_TEMP
        io: i
        field: DESC Over temperature
    '}
    bOverTemperature        : BOOL;
    {attribute 'pytmc' := '
        pv: REF_MARK
        io: i
        field: DESC Reference mark
    '}
    bReferenceMark          : BOOL;
    {attribute 'pytmc' := '
        pv: PHASED
        io: i
        field: DESC Is phased
    '}
    bIsPhased               : BOOL;
    {attribute 'pytmc' := '
        pv: FAULT
        io: i
        field: DESC Positioner fault
    '}
    bPositionerFault        : BOOL;
    {attribute 'pytmc' := '
        pv: AMP_ENABLED
        io: i
        field: DESC Amplifier enabled
    '}
    bAmplifierEnabled       : BOOL;
    {attribute 'pytmc' := '
        pv: IN_POSITION
        io: i
        field: DESC In position
    '}
    bInPosition             : BOOL;
    {attribute 'pytmc' := '
        pv: BRAKE_ENABLED
        io: i
        field: DESC Brake enabled
    '}
    bBrakeEnabled           : BOOL;
END_STRUCT
END_TYPE

// ---- DUTs/DS402/ST_DS402Drive.TcDUT
TYPE ST_DS402Drive:
STRUCT
    (* Global variables for the TPDO data from the drive. Each one is linked to the respective TPDO channel. *)
    stDriveStatus 			AT %I*	: 	ST_DS402DriveStatus;
    {attribute 'pytmc' := '
        pv: eOpModeDisplay
        io: i
        field: DESC MCS2 current operating mode
    '}
    nModeOfOperationDisplay AT %I*	: 	SINT;
    //nActualPosition 		AT %I*	: 	DINT;
    (*CSP drive mode*)
    nFollowingError 		AT %I*	: 	DINT;
    (* Global variables for the RPDO data to the drive. Each one is linked to the respective RPDO channel. *)
    // connected to I/O Task 'Control Word'
    nDriveControl			AT %Q*	:	UINT;
    // Connected to NC task Ctrl 1 and Ctrl 2
    nDriveControlNC			AT %I*	:	UINT;
    nTargetPosition 		AT %Q* 	: 	DINT;
    nModeOfOperation 		AT %Q* 	: 	SINT;
    nModeOfOperationNC 		AT %I* 	: 	SINT;
    (* Global variables for the RPDO data to the drive. Each one is linked to the respective RPDO channel. *)
    nProfilVelocity 		AT %Q* 	: 	DINT;
    nProfilAcceleration		AT %Q* 	: 	DINT;
    nProfilDecceleration	AT %Q* 	: 	DINT;
    nVelocityActualValue	AT %Q* 	: 	DINT;
    (* Global variables for the TPDO data from the drive. Each one is linked to the respective TPDO channel. *)
    nScantargetPosition		AT %Q*	: 	DINT;
    uScantargetVelocity		AT %Q*	: 	ULINT;
    (* Port Number of EtherCAT Slave *)
    nSlaveAddr	AT %I*  : UINT;
    (* EtherCAT slave ESM state, linked to the slave's InfoData.State.
       Low nibble is the state: 1=INIT, 2=PREOP, 4=SAFEOP, 8=OP. *)
    nEcatState	AT %I*  : UINT;
END_STRUCT
END_TYPE

// ---- DUTs/DS402/ST_MCS2ChanParameter.TcDUT
TYPE ST_MCS2ChanParameter :
STRUCT
    {attribute 'pytmc' := '
        pv: STEP_COUNT
        io: io
        field: DESC Open Loop Step Count
    '}
    nChanStep	: DINT := 500;

    {attribute 'pytmc' := '
        pv: STEP_EGU
        io: io
        field: DESC Step scale factor
    '}
    nChanStepEgu	: LREAL := 827.15;

    {attribute 'pytmc' := '
        pv: STEP_FREQ
        io: io
        field: DESC Step Frequency
    '}
    nChanStepFreq	: UINT := 500;

    {attribute 'pytmc' := '
        pv: STEP_VOLTAGE
        io: io
        field: DESC Step Amplitude
    '}
    nChanStepAmp	: UINT := 50;

    {attribute 'pytmc' := '
        pv: HOLD_TIME
        io: io
        field: DESC Close loop hold time
    '}
    nHoldTime	: UDINT := 30000;

    {attribute 'pytmc' := '
        pv: STEP_MOVE
        io: io
        field: ZNAM DISABLE
        field: ONAM ENABLE
        field: DESC Used to disable close loop mode
    '}
    bStepMoveCmd	: BOOL;

    {attribute 'pytmc' := '
        pv: STEP_FORWARD
        io: io
        field: DESC Jog one step count forward
    '}
    bStepForwardCmd	: BOOL;

    {attribute 'pytmc' := '
        pv: STEP_REVERSE
        io: io
        field: DESC Jog one step count backward
    '}
    bStepReverseCmd	: BOOL;

    {attribute 'pytmc' := '
        pv: MAX_CLF
        io: io
        field: DESC Max Close Loop Freq
    '}
    nMaxCloseLoopFreq     : UDINT;

    {attribute 'pytmc' := '
        pv: PTYPE
        io: io
        field: DESC Positioner Type
    '}
    nPositionerType	: UDINT;

    // Writable command pushed to 0x2004; the reader reads the drive value back
    // into it, so io:io serves both command and read-back on one symbol.
    {attribute 'pytmc' := '
        pv: CAL_OPT
        io: io
        field: DESC Calibration Options
    '}
    nCalibrationOpt       : DWORD;

    {attribute 'pytmc' := '
        pv: SENSOR_MODE
        io: io
        field: DESC Sensor Power Mode
    '}
    nSensorPowerMode      : UDINT;

    // Writable command pushed to 0x200B; the reader reads the drive value back
    // into it, so io:io serves both command and read-back on one symbol.
    {attribute 'pytmc' := '
        pv: REF_OPT
        io: io
        field: DESC Referencing Options
    '}
    nReferencingOpt       	   : DWORD;

    {attribute 'pytmc' := '
        pv: REF_TYPE
        io: i
        field: DESC Reference Type
    '}
    nReferenceType 	: UDINT;

    {attribute 'pytmc' := '
        pv: SAFE_DIR
        io: io
        field: ZNAM FORWARD
        field: ONAM BACKWARD
        field: DESC Safe direction (0x200C), Pre-Op
    '}
    nSafeDir	: BOOL;

    {attribute 'pytmc' := '
        pv: MOTOR_LOAD
        io: i
        field: DESC Motor Load
    '}
    nMotorLoad	: USINT;

    {attribute 'pytmc' := '
        pv: CHAN_TYPE
        io: io
        field: DESC Channel Type
    '}
    nChannelType          : UDINT;

    {attribute 'pytmc' := '
        pv: LSCO
        io: io
        field: DESC Logical Scale Offset
    '}
    nLogicalScaleOffset   : UDINT; // should LINT

    {attribute 'pytmc' := '
        pv: LSCI
        io: io
        field: DESC Logical Scale Inversion
    '}
    nLogicalScaleInv  	 : BOOL;

    {attribute 'pytmc' := '
        pv: DO_CALIB
        io: io
        field: DESC Calibrate command
    '}
    bCalibrationCmd : BOOL;

    // Desired drive operating mode (source of truth). Default is closed-loop (CSP) absolute motion.
    {attribute 'pytmc' := '
        pv: OPMODE_REQ
        io: o
        field: DESC DS402 op mode request (closed loop)
    '}
    eOpModeReq : E_MCS2OpModeReq := E_MCS2OpModeReq.CLOSED_LOOP;

    {attribute 'pytmc' := '
        pv: chanState
        io: i
        field: DESC Channel configuration parameters.
    '}
    stChannelState        : ST_ChannelState;

    {attribute 'pytmc' := '
        pv: HOME_MODE
        io: i
        field: DESC Vendor Homing Modes.
    '}
    eHomeMode			  : E_MCS2HomeMethod := E_MCS2HomeMethod.AutoMethod;

    {attribute 'pytmc' := '
        pv: CHANTEMP
        io: i
        field: DESC Channel Temperature
    '}
    nChannelTemp          : INT;

    {attribute 'pytmc' := '
        pv: MOVE_TYPE
        io: i
        field: DESC Movement Type
    '}
    nMovementType         : UDINT;

    {attribute 'pytmc' := '
        pv: BASE_UNIT
        io: i
        field: DESC Base Unit
    '}
    nBaseUnit             : UDINT;

    {attribute 'pytmc' := '
        pv: BASE_RES
        io: i
        field: DESC Base Resolution
    '}
    nBaseResolution       : DINT;

    {attribute 'pytmc' := '
        pv: DCIN
        io: io
        field: DESC Distance Code Inverted
    '}
    nDistCodeInv          : BOOL;

    {attribute 'pytmc' := '
        pv: POS_CTRL_OPT
        io: io
        field: DESC Positioner Control Options
    '}
    nPositionerCtrlOpt    : DWORD;

    {attribute 'pytmc' := '
        pv: ACT_MODE
        io: io
        field: DESC Actuator Mode
    '}
    nActuatorMode         : UDINT;

    {attribute 'pytmc' := '
        pv: MOTOR_LOAD_PROT
        io: io
        field: DESC Motor Load Protection Threshold
    '}
    nMotorLoadProt        : USINT;

    {attribute 'pytmc' := '
        pv: DIAG_CLF_MAX
        io: i
        field: DESC Diagnostic Closed Loop Frequency (max)
    '}
    nDiagClfMax           : UDINT;

    {attribute 'pytmc' := '
        pv: DIAG_CLF_AVG
        io: i
        field: DESC Diagnostic Closed Loop Frequency (avg)
    '}
    nDiagClfAvg           : UDINT;

    {attribute 'pytmc' := '
        pv: MCS2_ERR
        io: i
        field: DESC Last MCS2 drive error code (0x603F)
    '}
    nMCS2ErrorCode        : UINT;

    {attribute 'pytmc' := '
        pv: MCS2_ERR_MSG
        io: i
        field: DESC Decoded MCS2 drive error
    '}
    sMCS2ErrorMessage     : STRING;

    // Read-only decode of the drive's actual Referencing Options (REF_OPT,
    // 0x200B) into individual flags for verification. Command via REF_OPT.
    {attribute 'pytmc' := '
        pv: REF_OPT:START_DIR_BACK
        io: i
        field: DESC Ref start direction backward (bit0)
    '}
    bRefStartDirBackward  : BOOL;
    {attribute 'pytmc' := '
        pv: REF_OPT:REVERSE_DIR
        io: i
        field: DESC Ref reverse dir, multi-mark (bit1)
    '}
    bRefReverseDir        : BOOL;
    {attribute 'pytmc' := '
        pv: REF_OPT:AUTO_ZERO
        io: i
        field: DESC Ref auto-zero on reference found (bit2)
    '}
    bRefAutoZero          : BOOL;
    {attribute 'pytmc' := '
        pv: REF_OPT:ABORT_ENDSTOP
        io: i
        field: DESC Ref abort on end stop (bit3)
    '}
    bRefAbortOnEndStop    : BOOL;
    {attribute 'pytmc' := '
        pv: REF_OPT:CONT_ON_REF
        io: i
        field: DESC Ref continue on reference found (bit4)
    '}
    bRefContinueOnRefFound: BOOL;
    {attribute 'pytmc' := '
        pv: REF_OPT:STOP_ON_REF
        io: i
        field: DESC Ref stop on reference found (bit5)
    '}
    bRefStopOnRefFound    : BOOL;
    {attribute 'pytmc' := '
        pv: REF_OPT:INVALIDATE
        io: i
        field: DESC Ref invalidate is-ref flag (bit24)
    '}
    bRefInvalidate        : BOOL;

    // Read-only decode of the drive's actual Calibration Options (CAL_OPT,
    // 0x2004) into individual flags for verification. Command via CAL_OPT.
    {attribute 'pytmc' := '
        pv: CAL_OPT:DIR_BACK
        io: i
        field: DESC Calib move direction backward (bit0)
    '}
    bCalDirBackward       : BOOL;
    {attribute 'pytmc' := '
        pv: CAL_OPT:DETECT_DCI
        io: i
        field: DESC Calib detect dist code inv (bit1)
    '}
    bCalDetectDistCodeInv : BOOL;
    {attribute 'pytmc' := '
        pv: CAL_OPT:ADV_SENSOR
        io: i
        field: DESC Calib advanced sensor correction (bit2)
    '}
    bCalAdvSensorCorr     : BOOL;
    {attribute 'pytmc' := '
        pv: CAL_OPT:LIM_TRAVEL
        io: i
        field: DESC Calib limited travel, endstop (bit8)
    '}
    bCalLimitedTravelRange: BOOL;

    {attribute 'hide'}
    nHomeVeloFast         : UDINT;
    {attribute 'hide'}
    nSoftLimMin           : LINT;
    {attribute 'hide'}
    nSoftLimMax           : LINT;
    {attribute 'hide'}
    nHomeVeloSlow         : UDINT;
    {attribute 'hide'}
    nHomeAcc              : UDINT;
    {attribute 'hide'}
    nScaledFErrWin        : DINT;
    {attribute 'hide'}
    nHomeOffset           : DINT;
    {attribute 'hide'}
    nHomeMethod           : SINT;
    {attribute 'hide'}
    fScalingFactor		  : LREAL := 0.000001;
    {attribute 'hide'}
    fHomeAcc			  : LREAL := 0.8;
    // ====== Channel-specific object indices ======
    nSubIndex                : BYTE := 0;        // Main subindex (which channel)
    {attribute 'hide'}
    nChanFErrWinIdx          : WORD;
    {attribute 'hide'}
    nChanMotorLoadIdx        : WORD;
    {attribute 'hide'}
    nChanErrorCodeIdx        : WORD;
    {attribute 'hide'}
    nChanStepIdx             : WORD;
    {attribute 'hide'}
    nChanStepFreqIdx         : WORD;
    {attribute 'hide'}
    nChanStepAmpIdx          : WORD;
    {attribute 'hide'}
    nChanSoftLimitIdx        : WORD;
    {attribute 'hide'}
    nChanHomeOffsIdx         : WORD;
    {attribute 'hide'}
    nChanHomeMethodIdx       : WORD;
    {attribute 'hide'}
    nChanHomeVeloIdx         : WORD;
    {attribute 'hide'}
    nChanhomeAccIdx          : WORD;
    {attribute 'hide'}
    nCHanMaxCloseLoopFreqIdx : WORD;
    {attribute 'hide'}
    nChanPositionerTypeIdx   : WORD;
    {attribute 'hide'}
    nChanCalibrationOptIdx   : WORD;
    {attribute 'hide'}
    nChanSensorPowerModeIdx  : WORD;
    {attribute 'hide'}
    nChanReferencingOptIdx   : WORD;
    {attribute 'hide'}
    nChanReferenceTypeIdx    : WORD;
    {attribute 'hide'}
    nChanSafeDirIdx          : WORD;
    {attribute 'hide'}
    nChannelTypeIdx          : WORD;
    {attribute 'hide'}
    nChanStateIdx            : WORD;
    {attribute 'hide'}
    nChanLogicalScaleOfsIdx  : WORD;
    {attribute 'hide'}
    nChanLogicalScaleInvIdx  : WORD;
    {attribute 'hide'}
    nChanChannelTempIdx      : WORD;
    {attribute 'hide'}
    nChanMovementTypeIdx     : WORD;
    {attribute 'hide'}
    nChanBaseUnitIdx         : WORD;
    {attribute 'hide'}
    nChanBaseResolutionIdx   : WORD;
    {attribute 'hide'}
    nChanDistCodeInvIdx      : WORD;
    {attribute 'hide'}
    nChanPositionerCtrlOptIdx: WORD;
    {attribute 'hide'}
    nChanActuatorModeIdx     : WORD;
    {attribute 'hide'}
    nChanMotorLoadProtIdx    : WORD;
    {attribute 'hide'}
    nChanDiagClfIdx          : WORD;
    fPosition : LREAL;
    bStageReady : BOOL;
    // Temporary workaround: Avoid declaring mc_power externally from FB_MotionStage
    bOverrideDirEnable : BOOL := TRUE;
    bEnableHardwareOps : BOOL := TRUE;
    nReadTime : TIME := T#5S;
END_STRUCT
END_TYPE

// ---- DUTs/E_EpicsHomeCmd.TcDUT
{attribute 'qualified_only'}
{attribute 'strict'}
TYPE E_EpicsHomeCmd :
    // Defines the valid options for homing in FB_MotionStage
(
    LOW_LIMIT := 1, // Low limit switch
    HIGH_LIMIT := 2, // High limit switch
    HOME_VIA_LOW := 3, // Home switch via low switch
    HOME_VIA_HIGH := 4, // Home switch via high switch
    ABSOLUTE_SET := 15, // Set here to be fHomePosition
    // MCS2
    AutoMethod := -1, // DS402 Auto method; referencing routine set by positioner type
    CURRENT_POSITION_METHOD := 37,
    NONE := -99 // Do not home, ever
) := NONE;
END_TYPE

// ---- DUTs/ST_AxisParameterSetExposed.TcDUT
TYPE ST_AxisParameterSetExposed :
    // Collects the axis parameters that are intentionally exposed to EPICS.
STRUCT
    // Maximum Dynamics
    {attribute 'pytmc' := '
        pv: MaxVel
        io: i
        field: DESC Maximum commandable speed of the axis in EU/s.
    '}
    fVeloMaximum                : LREAL; // Maximum commandable speed of the axis in EU/s.
    {attribute 'pytmc' := '
        pv: MaxAccel
        io: i
        field: DESC Maximum rate of increase in speed of the axis in EU/s^2.
    '}
    fAccelerationMax            : LREAL; // Maximum rate of increase in speed of the axis in EU/s^2.
    {attribute 'pytmc' := '
        pv: MaxDecel
        io: i
        field: DESC Maximum rate of decrease in speed of the axis in EU/s^2.
    '}
    fDecelerationMax            : LREAL; // Maximum rate of decrease in speed of the axis in EU/s^2.

    // Monitoring
    {attribute 'pytmc' := '
        pv: PosLagEn
        io: i
        field: DESC TRUE if position lag monitor (also known as stall monitor) is enabled.
    '}
    bCtrlEnablePosDiffControl   : WORD;  // Enable/Disable state of Position Lag Monitor.
    {attribute 'pytmc' := '
        pv: PosLagVal
        io: i
        field: DESC Maximum magnitude of position lag in EU.
    '}
    fCtrlPosDiffMax             : LREAL; // Maximum magnitude of position lag in EU.
    {attribute 'pytmc' := '
        pv: PosLagTime
        io: i
        field: DESC Maximum allowable duration outside of maximum position lag value in seconds.
    '}
    fCtrlPosDiffMaxTime         : LREAL; // Maximum allowable duration outside of maximum position lag value in seconds.

    // Limit Switches
    {attribute 'pytmc' := '
        pv: SLimMinEn
        io: i
        field: DESC TRUE if controller static minimum limit is enabled.
    '}
    bEncEnableSoftEndMinControl : WORD;  // Enable/Disable state of controller static minimum limit.
    {attribute 'pytmc' := '
        pv: SLimMaxEn
        io: i
        field: DESC TRUE if controller static maximum limit is enabled.
    '}
    bEncEnableSoftEndMaxControl : WORD;  // Enable/Disable state of controller static maximum limit.
    {attribute 'pytmc' := '
        pv: SLimMin
        io: i
        field: DESC Minimum commandable position of the axis in EU.
    '}
    fEncSoftEndMin              : LREAL; // Minimum commandable position of the axis in EU.
    {attribute 'pytmc' := '
        pv: SLimMax
        io: i
        field: DESC Maximum commandable position of the axis in EU.
    '}
    fEncSoftEndMax              : LREAL; // Maximum commandable position of the axis in EU.

    // Encoder Evaluation
    {attribute 'pytmc' := '
        pv: EncScaling
        io: i
        field: DESC Encoder scaling numerator / denominator in EU/COUNT.
    '}
    fEncScaleFactorInternal      : LREAL; // Encoder scaling numerator / denominator in EU/COUNT.
    {attribute 'pytmc' := '
        pv: EncOffset
        io: i
        field: DESC Encoder offset in EU.
    '}
    fEncOffset                   : LREAL; // Encoder offset in EU.

END_STRUCT
END_TYPE

// ---- DUTs/E_LCLSMotionError.TcDUT
{attribute 'qualified_only'}
{attribute 'strict'}
TYPE E_LCLSMotionError :
(
    ABORTED := 16#7900,
    UNSAFE := 16#7901,
    INVALID := 16#7902,
    MCS2_FAULT := 16#7903,
    TEST := 16#FFFF
) UDINT;
END_TYPE

// ---- DUTs/E_MotionFFType.TcDUT
{attribute 'qualified_only'}
TYPE E_MotionFFType :
(
    STOPPER_FAULT := 16#1000,
    ZERO_RATE := 16#1001,
    BPTM_TIMEOUT := 16#1002,
    BPTM_ERROR := 16#1003,
    MAINT_MODE := 16#1004,
    NOT_A_STATE := 16#1005,
    INVALID_GOAL := 16#1006,
    TOO_MANY_TRIPS := 16#1007,
    BP_MISMATCH := 16#1008,
    INTERNAL_ERROR := 16#1009,
    PNEUMATIC_MOVE := 16#1010,
    MOT_GENERIC := 16#1011,
    LOW_RESERVED_NC := 16#2000,
    HIGH_RESERVED_NC := 16#20FF,
    DEVICE_MOVE := 16#2100
) UINT := MOT_GENERIC;
END_TYPE

// ---- DUTs/E_StatePMPSStatus.TcDUT
{attribute 'qualified_only'}
{attribute 'strict'}
TYPE E_StatePMPSStatus :
(
    // No other enum state describes it
    UNKNOWN := 0,
    // Moving toward a known state
    TRANSITION := 1,
    // Within a known state, not trying to leave
    AT_STATE := 2,
    // PMPS is in some way disabled, either with maint mode or arbiter disable
    DISABLED := 3
);
END_TYPE

// ---- DUTs/ST_MotionEpicsInterface.TcDUT
TYPE ST_MotionEpicsInterface :
    // Defines the EPICS interface to moving a motor in TwinCAT
STRUCT
 // Name to use for log messages, fast faults, etc.
    sName: STRING;
    // Set to gantry difference tolerance
    nGantryTol: LINT:=0;
    // Encoder count at which this axis is aligned with other axis
    nEncRef: ULINT:=0;

    (* Commands *)
    // Used internally to request enables
    bEnable: BOOL;

    // Used internally to reset errors and other state
    {attribute 'pytmc' := '
        pv: PLC:bReset
        io: io
        field: ZNAM FALSE
        field: ONAM TRUE
        field: DESC Used internally to reset errors
    '}
    bReset: BOOL;
    // Used internally and by the IOC to start or stop a move
    bExecute: BOOL;

    (* Command Args *)
    // Used internally and by the IOC to pick what kind of move to do
    nCommand: INT;
    // Used internally and by the IOC to pass additional data to some commands
    nCmdData: INT;
    // Used internally and by the IOC to pick a destination for the move
    fPosition: LREAL;
    // Used internally and by the IOC to pick a move velocity
    fVelocity: LREAL;
    // Used internally and by the IOC to pick a move acceleration
    fAcceleration: LREAL;
    // Used internally and by the IOC to pick a move deceleration
    fDeceleration: LREAL;
    // Used internally and by the IOC to pick a home position
    {attribute 'pytmc' := '
        pv: PLC:fHomePosition
        io: io
        field: DESC Used internally and by the IOC to pick home position
    '}
    fHomePosition: LREAL;

    (* Info *)
    // Unique ID assigned to each axis in the NC
    nMotionAxisID: UDINT:=0;
    (* Returns *)
    // TRUE if in the middle of a command
    bBusy: BOOL;
    // TRUE if we've done a command and it has finished
    bDone: BOOL;
    // TRUE if the motor has been homed, or does not need to be homed
    bHomed: BOOL;

    // TRUE if we're in an error state
    {attribute 'pytmc' := '
        pv: PLC:bError
        io: i
        field: ZNAM FALSE
        field: ONAM TRUE
        field: DESC TRUE if we are in an error state
        update: 100Hz notify
    '}
    bError: BOOL;
    // Error code if nonzero
    {attribute 'pytmc' := '
        pv: PLC:nErrorId
        io: i
        field: DESC Error code if nonzero
        update: 100Hz notify
    '}
    nErrorId: UDINT;
    // Message to identify the error state
    {attribute 'pytmc' := '
        pv: PLC:sErrorMessage
        io: i
        field: DESC Message to identify the error state
        update: 100Hz notify
    '}
    sErrorMessage: STRING;

    // Misc axis status information for the IOC
    stAxisStatus: tc2_mc2.ST_AxisStatus;
END_STRUCT
END_TYPE

// ---- DUTs/ST_MotionStage.TcDUT
TYPE ST_MotionStage :
    // Defines the EPICS interface to moving a motor in TwinCAT
STRUCT
    (* Hardware *)

    // PLC Axis Reference
    Axis: AXIS_REF;
    // NC Forward Limit Switch: TRUE if ok to move
    bLimitForwardEnable AT %I*: BOOL;
    // NC Backward Limit Switch: TRUE if ok to move
    bLimitBackwardEnable AT %I*: BOOL;
    // NO Home Switch: TRUE if at home
    bHome AT %I*: BOOL;
    // NC Brake Output: TRUE to release brake
    bBrakeRelease AT %Q*: BOOL;
    // NC STO Input: TRUE if ok to move
    {attribute 'pytmc' := '
        pv: PLC:bHardwareEnable
        io: i
        field: ZNAM FALSE
        field: ONAM TRUE
        field: DESC TRUE if STO not hit
    '}
    bHardwareEnable AT %I*: BOOL;

    // Raw encoder IO for ULINT (Biss-C)
    nRawEncoderULINT AT %I*: ULINT;
    // Raw encoder IO for UINT (Relative Encoders)
    nRawEncoderUINT AT %I*: UINT;
    // Raw encoder IO for INT (LVDT)
    nRawEncoderINT AT %I*: INT;
    // Raw encoder IO for INT (EL5072 LVDT)
    nRawEncoderDINT AT %I*: DINT;

    (* Psuedo-hardware *)

    // Forward enable EPS summary
    bAllForwardEnable: BOOL:=FALSE;
    // Backward enable EPS summary
    bAllBackwardEnable: BOOL:=FALSE;
    // Enable EPS summary encapsulating emergency stop button and any additional motion preventive hardware
    bAllEnable: BOOL:=FALSE;
    // Forward virtual gantry limit switch
    bGantryForwardEnable: BOOL:=FALSE;
    // Backward virtual gantry limit switch
    bGantryBackwardEnable: BOOL:=FALSE;
    // Encoder count summary, if linked above
    {attribute 'pytmc' := '
        pv: PLC:nEncoderCount
        io: i
        field: DESC Count from encoder hardware
    '}
    nEncoderCount: UDINT;
    // Forward Enable EPS struct
    {attribute 'pytmc' := '
        pv: PLC:stEPSF
        io: i
        field: DESC Forward Enable Interlocks
    '}
    stEPSForwardEnable: DUT_EPS;
    // Backward Enable EPS struct
    {attribute 'pytmc' := '
        pv: PLC:stEPSB
        io: i
        field: DESC Backward Enable Interlocks
    '}
    stEPSBackwardEnable: DUT_EPS;
    // Power Enable EPS struct
    {attribute 'pytmc' := '
        pv: PLC:stEPSP
        io: i
        field: DESC Power Interlocks
    '}
    stEPSPowerEnable: DUT_EPS;

    (* Settings *)
    // Name to use for log messages, fast faults, etc.
    sName: STRING;
    // If TRUE, we want to enable the motor independently of PMPS or other safety systems.
    bPowerSelf: BOOL:=FALSE;
    // Determines when we automatically enable the motor
    nEnableMode: E_StageEnableMode:=E_StageEnableMode.DURING_MOTION;
    // Determines when we automatically disengage the brake
    nBrakeMode: E_StageBrakeMode:=E_StageBrakeMode.IF_ENABLED;
    // Determines our encoder homing strategy
    nHomingMode: E_EpicsHomeCmd:=E_EpicsHomeCmd.NONE;
    // Set true to activate gantry EPS
    bGantryAxis: BOOL:=FALSE;

    // Set to gantry difference tolerance
    nGantryTol: LINT:=0;

    // Encoder count at which this axis is aligned with other axis
    nEncRef: ULINT:=0;

    (* Commands *)
    // Used internally to request enables
    bEnable: BOOL;
    // Used internally to reset errors and other state
    {attribute 'pytmc' := '
        pv: PLC:bReset
        io: io
        field: ZNAM FALSE
        field: ONAM TRUE
        field: DESC Used internally to reset errors
    '}
    bReset: BOOL;
    // Used internally and by the IOC to start or stop a move
    bExecute: BOOL;
    // Used by the IOC to disable an axis
    {attribute 'pytmc' := '
        pv: PLC:bUserEnable
        io: io
        field: ZNAM DISABLE
        field: ONAM ENABLE
        field: DESC Used to disable power entirely for an axis
        autosave_pass1: VAL
    '}
    bUserEnable: BOOL := 1;

    (* Shortcut Commands *)
    // Start a move to fPosition with fVelocity
    bMoveCmd: BOOL;
    // Start the homing routine
    {attribute 'pytmc' := '
        pv: PLC:bHomeCmd
        io: io
        field: DESC Start the homing routine
    '}
    bHomeCmd: BOOL;

    (* Command Args *)
    // Used internally and by the IOC to pick what kind of move to do
    nCommand: INT;
    // Used internally and by the IOC to pass additional data to some commands
    nCmdData: INT;
    // Used internally and by the IOC to pick a destination for the move
    fPosition: LREAL;
    // Used internally and by the IOC to pick a move velocity
    fVelocity: LREAL;
    // Used internally and by the IOC to pick a move acceleration
    fAcceleration: LREAL;
    // Used internally and by the IOC to pick a move deceleration
    fDeceleration: LREAL;
    // Used internally and by the IOC to pick a home position
    {attribute 'pytmc' := '
        pv: PLC:fHomePosition
        io: io
        field: DESC Used internally and by the IOC to pick home position
        autosave_pass1: VAL
    '}
    fHomePosition: LREAL;

    (* Info *)
    // Unique ID assigned to each axis in the NC
    nMotionAxisID: UDINT:=0;

    (* Returns *)
    // TRUE if done enabling
    bEnableDone: BOOL;
    // TRUE if in the middle of a command
    bBusy: BOOL;
    // TRUE if we've done a command and it has finished
    bDone: BOOL;
    // TRUE if the motor has been homed, or does not need to be homed
    bHomed: BOOL;
    // TRUE if we have safety permission to move
    bSafetyReady: BOOL;
    // TRUE if we're in an error state
    {attribute 'pytmc' := '
        pv: PLC:bError
        io: i
        field: ZNAM FALSE
        field: ONAM TRUE
        field: DESC TRUE if we are in an error state
    '}
    bError: BOOL;
    // Error code if nonzero
    {attribute 'pytmc' := '
        pv: PLC:nErrorId
        io: i
        field: DESC Error code if nonzero
    '}
    nErrorId: UDINT;
    // Message to identify the error state
    {attribute 'pytmc' := '
        pv: PLC:sErrorMessage
        io: i
        field: DESC Message to identify the error state
    '}
    sErrorMessage: STRING;
    // Internal hook for custom error messages
    sCustomErrorMessage: STRING;
    // MC_ReadParameterSet Output
    stAxisParameters: ST_AxisParameterSet;
    // NC parameters that are exposed with pytmc pragmas
    {attribute 'pytmc' := '
        pv: PLC:AxisPar
        io: i
        field: DESC Axis configuration parameters in the numerical controller.
    '}
    stAxisParametersExposed: ST_AxisParameterSetExposed;
    // True if we've updated stAxisParameters at least once
    bAxisParamsInit: BOOL;

    // Misc axis status information for the IOC
    stAxisStatus: DUT_AxisStatus_v0_01;

    (* Other status information for users of the IOC *)
    // Position lag difference
    {attribute 'pytmc' := '
        pv: PLC:fPosDiff
        io: i
        field: DESC Position lag difference
    '}
    fPosDiff: LREAL;

    (* Backlash compensation*)
    // Enabled axis backlash compensation
    {attribute 'pytmc' := '
        pv: PLC:bBacklashEn
        io: io
        field: ZNAM FALSE
        field: ONAM TRUE
        field: DESC Enable Backlash compensation
        autosave_pass1: VAL
    '}
    bUserBacklashEn: BOOL;

    // backlash compensation status
    {attribute 'pytmc' := '
        pv: PLC:bBacklasStatus
        io: i
        field: ZNAM DISABLED
        field: ONAM ENABLED
        field: DESC Backlash compensation status
    '}
    bBacklashStatus: BOOL;

    // Backlash compensation value
    {attribute 'pytmc' := '
        pv: PLC:fBacklash
        io: io
        field: DESC Backlash compensation
        autosave_pass1: VAL
    '}
    fBacklash: LREAL;

    // Current Backlash compensation value ?
    {attribute 'pytmc' := '
        pv: PLC:fCurrentBacklash
        io: i
        field: DESC Currently applied compensation
    '}
    fCurrentBacklash: LREAL;

    bRestoreDone : BOOL;
END_STRUCT
END_TYPE

// ---- DUTs/ST_PositionState.TcDUT
TYPE ST_PositionState :
    // Defines settings and current safety status for moves to specific positions for an axis
STRUCT
    // Name as queried via the NAME PV in EPICS
    {attribute 'pytmc' := '
        pv: NAME
        io: input
        field: DESC Name of this position state
    '}
    sName: STRING := 'Invalid';

    // Position associated with this state
    {attribute 'pytmc' := '
        pv: SETPOINT
        io: io
        field: DESC Axis position associated with this state
    '}
    fPosition: LREAL;

    {attribute 'pytmc' := '
        pv: ENCODER
        io: i
        field: DESC Encoder count associated with this state
    '}
    nEncoderCount: UDINT;

    // Maximum allowable deviation from fPosition while at the state
    fDelta: LREAL;

    // Speed at which to move to this state
    {attribute 'pytmc' := '
        pv: VELO
        io: io
        field: DESC Speed at which to move to this state
    '}
    fVelocity: LREAL;

    // (optional) Acceleration to use for moves to this state
    fAccel: LREAL;

    // (optional) Deceleration to use for moves to this state
    fDecel: LREAL;

    // Safety parameter. This must be set to TRUE by the PLC program to allow moves to this state. This is expected to change as conditions change.
    {attribute 'pytmc' := '
        pv: MOVE_OK
        io: i
        field: ZNAM FALSE
        field: ONAM TRUE
        field: DESC TRUE if the move would be safe
    '}
    bMoveOk: BOOL;

    // Signifies to FB_PositionStateLock that this state should be immutable
    bLocked: BOOL;

    // Set this to TRUE when you make your state. This defaults to FALSE so that uninitialized states can never be moved to
    bValid: BOOL;

    // Set this to TRUE when you want to use the raw encoder counts to define the state
    bUseRawCounts: BOOL;

    // Is set to TRUE by FB_PositionStateInternal when called
    bUpdated: BOOL;

    // We give this a state name and it is used to load parameters from the pmps database.
    stPMPS: ST_DbStateParams;
	
	// Set this to TRUE to enable use of the iSequence value to sequence moves that incorporate this state.
    {attribute 'pytmc' := '
        pv: SEQUENCE_MOVES
        io: i
        field: DESC TRUE if this state represents a state intended to be moved in sequence with other axes
    '}
	bSequenceMoves: BOOl;
	
	// Set this value to the sequence number that you want this state to have relative to other axes.
	// E.g. if this state has iSequence = 2 and it is being moved with a state with iSequence = 1, then
	// the iSequence = 1 state will be moved first and this state will only be moved after.
    {attribute 'pytmc' := '
        pv: SEQUENCE_ORDER
        io: i
        field: DESC Relative sequence order for the axis movement corresponding to this state.
    '}
	iSequenceOrder: UINT := 1;
END_STRUCT
END_TYPE

// ---- DUTs/ST_StateEpicsToPlc.TcDUT
TYPE ST_StateEpicsToPlc :
(*
    This data structure contains the standard EPICS input connection points for the state movers.

    The data in this struct flows from EPICS to the PLC.

    It includes everything except the SET PV, which cannot be included here
    as it is sourced from enum values unique to the application, and the PMPS PVs, which are
    gathered in their own data type, ST_StatePMPSEpicsToPlc. That actually means that this only
    holds the RESET PV, for now.

    nSetValue here is actively used by state blocks even though it is not exposed
    directly to EPICS. You should avoid manually modifying it or else
    you may interfere with normal operations of the state function blocks.

    For including your own ENUM input, you should pytmc pragma the PV name to end in "SET",
    and match the prefix of this FB's "RESET" PV. Then, you can include your enum
    as the eEnumSet IN_OUT var and let the EPICS IOC handle it.
*)
STRUCT
    // For internal use only. This holds new goal positions as an integer, else it is 0 if there is no new state move request. It is written to from the user's input enum.
    nSetValue: UINT;

    // Set this to TRUE to acknowledge and clear an error.
    {attribute 'pytmc' := '
        pv: RESET
        io: io
        field: ZNAM False
        field: ONAM True
    '}
    bReset: BOOL;
END_STRUCT
END_TYPE

// ---- DUTs/ST_StatePlcToEpics.TcDUT
TYPE ST_StatePlcToEpics :
(*
    This data structure contains the standard EPICS connection points for the state movers.

    The data in this struct flows from the PLC to EPICS.

    It includes everything except the GET PV, which cannot be included here
    as it is sourced from enum values unique to the application, and the PMPS PVs, which are
    gathered in their own data type, ST_StatePMPSPlcToEpics.

    nGetValue here is actively used by state blocks even though it is not exposed directly
    to EPICS. It is safe to read this value, but you should avoid modifying it, which may
    interfere with normal operations of the state function blocks.

    For including your own ENUM input, you should pytmc pragma the PV name to end in "GET",
    and match the prefix of this FB's "DONE" PV. Then, you can include your enum
    as the eEnumGet IN_OUT var and let the EPICS IOC handle it.
*)
STRUCT
    // For internal use only. This holds the current position index as an integer, else it is 0 if we are changing states or not at any particular state.
    nGetValue: UINT;
    // This will be TRUE when we are in an active state move and FALSE otherwise.
    {attribute 'pytmc' := '
        pv: BUSY
        io: i
        field: ZNAM False
        field: ONAM True
    '}
    bBusy: BOOL;
    // This will be TRUE after a move completes and FALSE otherwise.
    {attribute 'pytmc' := '
        pv: DONE
        io: i
        field: ZNAM False
        field: ONAM True
    '}
    bDone: BOOL;
    // This will be TRUE if the most recent move had an error and FALSE otherwise.
    {attribute 'pytmc' := '
        pv: ERR
        io: i
        field: ZNAM False
        field: ONAM True
    '}
    bError: BOOL;
    // This will be set to an NC error code during an error if one exists or left at 0 otherwise.
    {attribute 'pytmc' := '
        pv: ERRID
        io: i
    '}
    nErrorID: UDINT;
    // This will be set to an appropriate error message during an error if one exists or left as an empty string otherwise.
    {attribute 'pytmc' := '
        pv: ERRMSG
        io: i
    '}
    sErrorMsg: STRING;
END_STRUCT
END_TYPE

// ---- DUTs/ST_StatePMPSEpicsToPlc.TcDUT
TYPE ST_StatePMPSEpicsToPlc :
(*
    This data structure contains the standard PMPS EPICS connection points for the state movers.

    The data in this struct flows from EPICS to the PLC.
*)
STRUCT
    // User setting: TRUE to enable the arbiter, FALSE to disable it.
    {attribute 'pytmc' := '
        pv: PMPS:ARB:ENABLE
        io: io
    '}
    bArbiterEnabled: BOOL := TRUE;
    // User setting: TRUE to enable maintenance mode (Fast fault, free motion), FALSE to disable it.
    {attribute 'pytmc' := '
        pv: PMPS:MAINT
        io: io
    '}
    bMaintMode: BOOL;
END_STRUCT
END_TYPE

// ---- DUTs/ST_EL5042_Status.TcDUT
TYPE ST_EL5042_Status :
STRUCT
END_STRUCT
END_TYPE

// ---- DUTs/E_EpicsInOut.TcDUT
{attribute 'qualified_only'}
// Example EPICS states enum for use in all versions of the states FBs
// Remove strict attribute for easier handling
TYPE E_EpicsInOut :
(
    UNKNOWN := 0, // UNKNOWN must be in slot 0 or the FB breaks
    OUT := 1, // OUT at slot 1 is a convention
    IN := 2
) UINT;
END_TYPE

// ---- DUTs/E_EpicsMotorCmd.TcDUT
{attribute 'qualified_only'}
{attribute 'strict'}
TYPE E_EpicsMotorCmd :
    // Defines valid EPICS commands for nCommand
(
    JOG := 0,
    MOVE_VELOCITY := 1,
    MOVE_RELATIVE := 2,
    MOVE_ABSOLUTE := 3,
    MOVE_MODULO := 4,
    HOME := 10,
    GEAR := 30,
    CALIBRATE:=40
);
END_TYPE

// ---- DUTs/E_MotionRequest.TcDUT
{attribute 'qualified_only'}
{attribute 'strict'}
TYPE E_MotionRequest :
    // Defines behavior options for when FB_MotionRequest is run during an active move from another source
(
    WAIT := 0,
    INTERRUPT := 1,
    ABORT := 2
);
END_TYPE

// ---- DUTs/E_StageBrakeMode.TcDUT
{attribute 'qualified_only'}
{attribute 'strict'}
TYPE E_StageBrakeMode :
    // Defines when to send the brake disengage signal in FB_MotionStage
(
    IF_ENABLED, // Disengage brake when the motor is enabled
    IF_MOVING, // Disengage brake when the motor is moving
    NO_BRAKE // Do not change the brake state in FB_MotionStage
);
END_TYPE

// ---- DUTs/E_StageEnableMode.TcDUT
{attribute 'qualified_only'}
{attribute 'strict'}
TYPE E_StageEnableMode :
    // Define conditions when FB_MotionStage automatically sets bEnable
(
    ALWAYS, // Always set bEnable to TRUE
    NEVER,  // Only change bEnable on errors
    DURING_MOTION  // Enable before motion, disable after motion
);
END_TYPE

// ---- DUTs/ST_MotionPneumaticActuator.TcDUT
{attribute 'qualified_only'}
{attribute 'strict'}
TYPE ST_MotionPneumaticActuator :
    // Defines the EPICS interface to actuating a pneumatic stage
STRUCT
     (* Hardware *)
    //Readbacks
    //Limit Switch
    {attribute 'pytmc' := '
     pv: PLC:bInLimitSwitch
     io: i
     field: ZNAM FALSE
     field: ONAM TRUE
     field: DESC TRUE if IN limit is reached
    '}
    i_bInLimitSwitch    :    BOOL;
    {attribute 'pytmc' := '
     pv: PLC:bOutLimitSwitch
     io: i
     field: ZNAM FALSE
     field: ONAM TRUE
     field: DESC TRUE if OUT limit is reached
    '}
    i_bOutLimitSwitch    :    BOOL;
    //Controls
    //Digital outputs
    {attribute 'pytmc' := '
    pv: bRetractDigitalOutput;
    io: i;
    field: ONAM FALSE
    field: ZNAM TRUE
    field: DESC TRUE if Retract digital output is active
    '}
    q_bRetract    :    BOOL;
    {attribute 'pytmc' := '
    pv: bInsertDigitalOutput;
    io: i;
    field: ONAM FALSE
    field: ZNAM TRUE
    field: DESC TRUE if Insert digital output is active
    '}
    q_bInsert    :    BOOL;


    //Logic and supervisory
    {attribute 'pytmc' := '
    pv: bInterlockOK;
    io: i;
    field: ZNAM FALSE
    field: ONAM TRUE
    field: DESC True if the actuator has permission to move in either direction
    '}
    bILK_OK: BOOL;
    {attribute 'pytmc' := '
    pv: bInsertEnable;
    io: i;
    field: ZNAM FALSE
    field: ONAM TRUE
    field: DESC True if the actuator had permission to be retracted
    '}
    bInsertOK    :    BOOL;
    {attribute 'pytmc' := '
    pv: bRetractEnable;
    io: i;
    field: ZNAM FALSE
    field: ONAM TRUE
    field: DESC True if the actuator had permission to be inserted
    '}
    bRetractOK    :    BOOL;

    (* Commands *)
    // Used from Epics to comand the actuator to  move
    {attribute 'pytmc' := '
    pv: CMD:IN;
    io: io;
    field: DESC Used by EPICS and internally to request Insert motion
    '}
    bInsert_SW        :    BOOL;
    {attribute 'pytmc' := '
    pv: CMD:OUT;
    io: io;
    field: DESC Used by EPICS and internally to request retract motion
    '}
    bRetract_SW    :    BOOL;

    (*Returns*)
     // TRUE if in the middle of a command
    {attribute 'pytmc' := '
     pv: bBusy
     io: i
     field: ONAM FALSE
     field: ZNAM TRUE
     field: DESC TRUE if in the middle of a command
    '}
    bBusy: BOOL;
    // TRUE if we've done a command and it has finished
    {attribute 'pytmc' := '
     pv: bDone
     io: i
     field: ONAM FALSE
     field: ZNAM TRUE
      field: DESC TRUE if command finished successfully
    '}
    bDone: BOOL;
     {attribute 'pytmc' := '
        pv: bReset
        io: io
        field: ZNAM FALSE
        field: ONAM TRUE
        field: DESC Used internally to reset errors
    '}
    bReset: BOOL;
    // TRUE if we're in an error state
    {attribute 'pytmc' := '
     pv: PLC:bError
     io: i
     field: ONAM FALSE
     field: ZNAM TRUE
     field: DESC TRUE if we're in an error state
    '}
    bError: BOOL;

     // Error code if nonzero
    {attribute 'pytmc' := '
     pv: PLC:nErrorId
     io: i
     field: DESC Error code if nonzero
    '}
    nErrorId: UDINT;
    // Message to identify the error state
    {attribute 'pytmc' := '
     pv: PLC:sErrorMessage
     io: i
     field: DESC Message to identify the error state
    '}
    sErrorMessage: STRING;
    {attribute 'pytmc' := '
    pv: nPositionState ;
    type: mbbi ;
    field: ZRST RETRACTED ;
    field: ONST INSERTED ;
    field: TWST MOVING ;
    field: THST INVALID ;
    io: i
    field: DESC Pneumatic actuator position
    '}

    eState    :    E_PnuematicActuatorPositionState := E_PnuematicActuatorPositionState.INVALID;

END_STRUCT
END_TYPE

// ---- DUTs/E_PnuematicActuatorPositionState.TcDUT
{attribute 'qualified_only'}
{attribute 'strict'}
// Defines the positions for a pnuematic actuator
TYPE E_PnuematicActuatorPositionState :
(
   RETRACTED    := 0, // Out limit switch is active
   INSERTED    := 1, // In limit switch is active
   MOVING    := 2, // Neither limit switches is Active
   INVALID :=3 // Invalid state
);
END_TYPE

// ---- DUTs/ST_RenishawAbsEnc.TcDUT
// Renishaw BiSS-C absolute encoder used with an EL5042
TYPE ST_RenishawAbsEnc :
STRUCT
    Count AT %I*: ULINT; // Connect to encoder "Position" input
    Status: ST_EL5042_Status; // Status struct placeholder
    Ref: ULINT; // Encoder zero position (useful for aligned position with gantries)
END_STRUCT
END_TYPE

// ---- DUTs/ST_StatePMPSPlcToEpics.TcDUT
TYPE ST_StatePMPSPlcToEpics :
(*
    This data structure contains the standard PMPS EPICS connection points for the state movers.

    The data in this struct flows from the PLC to EPICS.
*)
STRUCT
    // The database entry for the transition state. This should always be present.
    {attribute 'pytmc' := '
        pv: PMPS:TRANS
        io: i
    '}
    stTransitionDb: ST_DbStateParams;
END_STRUCT
END_TYPE

// ---- Tests/Helpers/E_TestStates.TcDUT
{attribute 'qualified_only'}
{attribute 'strict'}
TYPE E_TestStates :
(
    Unknown := 0,
    OUT := 1,
    TARGET1 := 2,
    TARGET2 := 3
) UINT;
END_TYPE

// ---- GVLs/MOTION_GVL.TcGVL
{attribute 'qualified_only'}
VAR_GLOBAL
    // Global file reader instance, used in fbStandardPMPSDB
    fbPmpsFileReader: FB_JsonFileToJsonDoc;
    {attribute 'pytmc' := '
        pv: @(PREFIX)DB
        io: io
    '}
    // Global DB handler, Must be called in PLC project to use the PMPS DB for a motion project
    fbStandardPMPSDB: FB_Standard_PMPSDB;
    // Debug, records the highest number of motors used in an ND states block in the PLC. Can be used to limit MotionConstants.MAX_STATE_MOTORS to save on memory usage and PV count.
    nMaxStateMotorCount: UINT;
    // Debug, records the highest state count in the PLC. Can be used to limit GeneralConstants.MAX_STATES to save on memory usage and PV count.
    nMaxStates: UINT;
END_VAR

// ---- GVLs/MotionConstants.TcGVL
{attribute 'qualified_only'}
(*
    Global Configurable Motion Constants

    These are reconfigurable at the project level.
    When reconfigured they are set prior to compilation and cannot be changed at runtime.
*)
VAR_GLOBAL CONSTANT
    (*
    Arbitary cap on multidimensional states to simplify statements for the compiler.
    This is reconfigurable at the project level and should be set to the highest number of motors used in a states block.
    If you are not sure how many motors are used per state block, check MOTION_GVL.nMaxStateMotorCount
    *)
    MAX_STATE_MOTORS: UINT := 3;
END_VAR

// ---- Tests/PRG_TEST.TcPOU
PROGRAM PRG_TEST
VAR
    fb_AtPositionState_Test: FB_AtPositionState_Test;
    fb_AxisParameterSetExposed_Test: FB_AxisParameterSetExposed_Test;
    fb_MiscStatesErrorFFO_Test: FB_MiscStatesErrorFFO_Test;
    fb_MotionBPTM_Test: FB_MotionBPTM_Test;
    fb_MotionClearAsserts_Test: FB_MotionClearAsserts_Test;
    fb_MotionReadPMPSDBND_Test: FB_MotionReadPMPSDBND_Test;
    fbMotionVirtualFrameTest: FB_MotionVirtualFrame_Test;
    fb_TestHelperSetAndMove_Test: FB_TestHelperSetAndMove_Test;
    fb_PositionStateRead_Test: FB_PositionStateRead_Test;
    fb_PositionStateReadND_Test: FB_PositionStateReadND_Test;
    fb_PositionStateMove_Test: FB_PositionStateMove_Test;
    fb_PositionStateMoveND_Test: FB_PositionStateMoveND_Test;
    fb_PositionStateND_Test: FB_PositionStateND_Test;
    fb_NCErrorFFO_Test: FB_NCErrorFFO_Test;
    fb_StatePMPSEnables_Test: FB_StatePMPSEnables_Test;
    fb_PerMotorFFOND_Test: FB_PerMotorFFOND_Test;
    fb_StatePMPSEnablesND_Test: FB_StatePMPSEnablesND_Test;
    fb_PositionStatePMPSND_Test: FB_PositionStatePMPSND_Test;
    fb_StateSetupHelper_Test: FB_StateSetupHelper_Test;
    fb_TestStateInitTiming: FB_TestStateInitTiming;
    fb_PowerEnableMode_Test: FB_PowerEnableMode_Test;
    fb_MotionBacklashCompensation_Test: FB_MotionBacklashCompensation_Test;
    fb_MCS2DriveManager_Test: FB_MCS2DriveManager_Test;
END_VAR


TcUnit.RUN();

END_PROGRAM

// ---- Tests/FB_AtPositionState_Test.TcPOU
FUNCTION_BLOCK FB_AtPositionState_Test EXTENDS TcUnit.FB_TestSuite
(*
    Test the following related helper functions:
    - F_PosOverLowerBound
    - F_PosUnderUpperBound
    - F_PosWithinDelta
    - F_AtPositionState
*)
VAR
    // For the multi-cycle tests
    stMotionStage: ST_MotionStage;
    fbMotionStage: FB_MotionStage;
    fbTestMove: FB_TestHelperSetAndMove;
    stPositionStateInactive: ST_PositionState;
    stPositionStateInvalid: ST_PositionState;
    stPositionStateGood: ST_PositionState;
    tonInactive: TON;
    fbInternalGood: FB_PositionStateInternal;
    fbInternalInvalid: FB_PositionStateInternal;
    nTestCounter: UINT;
    bOneTestDone: BOOL;
END_VAR


// Single cycle tests
TestPosOverLowerBoundYes();
TestPosOverLowerBoundNo();
TestPosUnderUpperBoundYes();
TestPosUnderUpperBoundNo();
TestPosWithinDeltaTooLow();
TestPosWithinDeltaTooHigh();
TestPosWithinDeltaJustRight();

// Multi cycle tests
fbMotionStage(stMotionStage:=stMotionStage);
stPositionStateInactive.sName := 'Inactive';
stPositionStateInactive.fPosition := 30.0;
stPositionStateInactive.fDelta := 1.0;
stPositionStateInactive.bValid := TRUE;
tonInactive(
    IN:=TRUE,
    PT:=T#1s,
);
TestAtPositionStateWithoutInternal();

stPositionStateInvalid.sName := 'Invalid';
stPositionStateInvalid.fPosition := 40.0;
stPositionStateInvalid.fDelta := 1.0;
stPositionStateInvalid.bValid := FALSE;
fbInternalInvalid(
    stMotionStage:=stMotionStage,
    stPositionState:=stPositionStateInvalid,
);
TestAtPositionStateInvalid();

stPositionStateGood.sName := 'Good';
stPositionStateGood.fPosition := 50.0;
stPositionStateGood.fDelta := 1.0;
stPositionStateGood.bValid := TRUE;
fbInternalGood(
    stMotionStage:=stMotionStage,
    stPositionState:=stPositionStateGood,
);
TestAtPositionStateTooLow();
TestAtPositionStateTooHigh();
TestAtPositionStateJustRight();
TestAtPositionStateTweak();
TestAtPositionStateLeave();

IF bOneTestDone THEN
    bOneTestDone := FALSE;
    nTestCounter := nTestCounter + 1;
    fbTestMove(
        stMotionStage:=stMotionStage,
        bExecute:=FALSE,
    );
END_IF

METHOD PRIVATE TestAtPositionStateInvalid
(*
    If a position state is invalid, it is never the right state.
*)
VAR

END_VAR

TEST('TestAtPositionStateInvalid');
IF nTestCounter <> 1 THEN
    RETURN;
END_IF

fbTestMove(
    stMotionStage:=stMotionstage,
    bExecute:=TRUE,
    fStartPosition:=stPositionStateInvalid.fPosition,
    fGoalPosition:=stPositionStateInvalid.fPosition,
);
IF fbTestMove.tElapsed > T#1s OR (stPositionStateInvalid.bUpdated AND fbTestMove.bSetDone) THEN
    AssertFalse(
        Condition:=F_AtPositionState(
            stMotionStage:=stMotionStage,
            stPositionState:=stPositionStateInvalid,
        ),
        Message:='Invalid state was marked OK',
    );
    AssertFalse(
        Condition:=fbTestMove.tElapsed > T#1s,
        Message:='Timeout in multi cycle test',
    );
    bOneTestDone := TRUE;
    TEST_FINISHED();
END_IF
END_METHOD

METHOD PRIVATE TestAtPositionStateJustRight
VAR
    fLocalGoal: LREAL;
END_VAR

TEST('TestAtPositionStateJustRight');
IF nTestCounter <> 4 THEN
    RETURN;
END_IF

fLocalGoal := stPositionStateGood.fPosition + 0.2*stPositionStateGood.fDelta;
fbTestMove(
    stMotionStage:=stMotionstage,
    bExecute:=TRUE,
    fStartPosition:=fLocalGoal,
    fGoalPosition:=fLocalGoal,
);
IF fbTestMove.tElapsed > T#1s OR (stPositionStateGood.bUpdated AND fbTestMove.bSetDone) THEN
    AssertTrue(
        Condition:=F_AtPositionState(
            stMotionStage:=stMotionStage,
            stPositionState:=stPositionStateGood,
        ),
        Message:='Within delta counted as outside range',
    );
    AssertFalse(
        Condition:=fbTestMove.tElapsed > T#1s,
        Message:='Timeout in multi cycle test',
    );
    bOneTestDone := TRUE;
    TEST_FINISHED();
END_IF
END_METHOD

METHOD PRIVATE TestAtPositionStateLeave
(*
    A move away from a state should be not at the state, even before we've left
*)
VAR
END_VAR

TEST('TestAtPositionStateLeave');
IF nTestCounter <> 6 THEN
    RETURN;
END_IF

fbTestMove(
    stMotionStage:=stMotionStage,
    bExecute:=TRUE,
    fStartPosition:=stPositionStateGood.fPosition,
    fGoalPosition:=stPositionStateGood.fPosition + 100 * stPositionStateGood.fDelta,
    fVelocity:=0.001,
    bHWEnable:=TRUE,
);

IF fbTestMove.tElapsed > T#5s OR (stPositionStateGood.bUpdated AND fbTestMove.bMotionStarted) THEN
    AssertTrue(
        Condition:=fbTestMove.fActPosition < stPositionStateGood.fPosition + stPositionStateGood.fDelta,
        Message:='We must be at the state location still to properly run this test.',
    );
    AssertFalse(
        Condition:=F_AtPositionState(
            stMotionStage:=stMotionStage,
            stPositionState:=stPositionStateGood,
        ),
        Message:='Leaving state is not at state once the move starts',
    );
    AssertFalse(
        Condition:=fbTestMove.tElapsed > T#5s,
        Message:='Timeout in multi cycle test',
    );
    bOneTestDone := TRUE;
    TEST_FINISHED();
END_IF
END_METHOD

METHOD PRIVATE TestAtPositionStateTooHigh
VAR
    fLocalGoal: LREAL;
END_VAR

TEST('TestAtPositionStateTooHigh');
IF nTestCounter <> 3 THEN
    RETURN;
END_IF

fLocalGoal := stPositionStateGood.fPosition + 2*stPositionStateGood.fDelta;
fbTestMove(
    stMotionStage:=stMotionstage,
    bExecute:=TRUE,
    fStartPosition:=fLocalGoal,
    fGoalPosition:=fLocalGoal,
);
IF fbTestMove.tElapsed > T#1s OR (stPositionStateGood.bUpdated AND fbTestMove.bSetDone) THEN
    AssertFalse(
        Condition:=F_AtPositionState(
            stMotionStage:=stMotionStage,
            stPositionState:=stPositionStateGood,
        ),
        Message:='Above delta counted as in range',
    );
    AssertFalse(
        Condition:=fbTestMove.tElapsed > T#1s,
        Message:='Timeout in multi cycle test',
    );
    bOneTestDone := TRUE;
    TEST_FINISHED();
END_IF
END_METHOD

METHOD PRIVATE TestAtPositionStateTooLow
VAR
    fLocalGoal: LREAL;
END_VAR

TEST('TestAtPositionStateTooLow');
IF nTestCounter <> 2 THEN
    RETURN;
END_IF

fLocalGoal := stPositionStateGood.fPosition - 2*stPositionStateGood.fDelta;
fbTestMove(
    stMotionStage:=stMotionstage,
    bExecute:=TRUE,
    fStartPosition:=fLocalGoal,
    fGoalPosition:=fLocalGoal,
);
IF fbTestMove.tElapsed > T#1s OR (stPositionStateGood.bUpdated AND fbTestMove.bSetDone) THEN
    AssertFalse(
        Condition:=F_AtPositionState(
            stMotionStage:=stMotionStage,
            stPositionState:=stPositionStateGood,
        ),
        Message:='Below delta counted as in range',
    );
    AssertFalse(
        Condition:=fbTestMove.tElapsed > T#1s,
        Message:='Timeout in multi cycle test',
    );
    bOneTestDone := TRUE;
    TEST_FINISHED();
END_IF
END_METHOD

METHOD PRIVATE TestAtPositionStateTweak
(*
    A small tweak move within the delta of a position state should be OK
*)
VAR

END_VAR

TEST('TestAtPositionStateTweak');
IF nTestCounter <> 5 THEN
    RETURN;
END_IF

fbTestMove(
    stMotionStage:=stMotionStage,
    bExecute:=TRUE,
    fStartPosition:=stPositionStateGood.fPosition,
    fGoalPosition:=stPositionStateGood.fPosition + 0.9 * stPositionStateGood.fDelta,
    fVelocity:=0.001,
    bHWEnable:=TRUE,
);

IF fbTestMove.tElapsed > T#5s OR (stPositionStateGood.bUpdated AND fbTestMove.bMotionStarted) THEN
    AssertTrue(
        Condition:=F_AtPositionState(
            stMotionStage:=stMotionStage,
            stPositionState:=stPositionStateGood,
        ),
        Message:='Small tweak in range should count as at state',
    );
    AssertFalse(
        Condition:=fbTestMove.tElapsed > T#5s,
        Message:='Timeout in multi cycle test',
    );
    bOneTestDone := TRUE;
    TEST_FINISHED();
END_IF
END_METHOD

METHOD PRIVATE TestAtPositionStateWithoutInternal
(*
    If a position state is never updated by the internal FB, it is never the right state.
*)
VAR

END_VAR

TEST('TestAtPositionStateWithoutInternal');
IF nTestCounter <> 0 THEN
    RETURN;
END_IF

fbTestMove(
    stMotionStage:=stMotionstage,
    bExecute:=TRUE,
    fStartPosition:=stPositionStateInactive.fPosition,
    fGoalPosition:=stPositionStateInactive.fPosition,
);
IF fbTestMove.tElapsed > T#1s OR (stPositionStateInvalid.bUpdated AND fbTestMove.bSetDone) THEN
    // Check for a different state to be bUpdated for timing purposes, this one never gets bUpdated
    AssertFalse(
        Condition:=F_AtPositionState(
            stMotionStage:=stMotionStage,
            stPositionState:=stPositionStateInactive,
        ),
        Message:='This is the control group, internal was not run so this should not work',
    );
    AssertFalse(
        Condition:=fbTestMove.tElapsed > T#1s,
        Message:='Timeout in multi cycle test',
    );
    bOneTestDone := TRUE;
    TEST_FINISHED();
END_IF
END_METHOD

METHOD PRIVATE TestPosOverLowerBoundNo
VAR
    stPositionState: ST_PositionState;
END_VAR

TEST('TestPosOverLowerBoundNo');
stPositionState.fPosition := 10;
stPositionState.fDelta := 1;

AssertFalse(
    Condition:=F_PosOverLowerBound(
        fPosition:=8.5,
        stPositionState:=stPositionState,
    ),
    Message:='Decided 8.5 > 9.0',
);
TEST_FINISHED();
END_METHOD

METHOD PRIVATE TestPosOverLowerBoundYes
VAR
    stPositionState: ST_PositionState;
END_VAR

TEST('TestPosOverLowerBoundYes');
stPositionState.fPosition := 10;
stPositionState.fDelta := 1;

AssertTrue(
    Condition:=F_PosOverLowerBound(
        fPosition:=9.1,
        stPositionState:=stPositionState,
    ),
    Message:='Decided 9.0 > 9.1',
);
TEST_FINISHED();
END_METHOD

METHOD PRIVATE TestPosUnderUpperBoundNo
VAR
    stPositionState: ST_PositionState;
END_VAR

TEST('TestPosUnderUpperBoundNo');
stPositionState.fPosition := 10;
stPositionState.fDelta := 1;

AssertFalse(
    Condition:=F_PosUnderUpperBound(
        fPosition:=12.0,
        stPositionState:=stPositionState,
    ),
    Message:='Decided 11.0 > 12.0',
);
TEST_FINISHED();
END_METHOD

METHOD PRIVATE TestPosUnderUpperBoundYes
VAR
    stPositionState: ST_PositionState;
END_VAR

TEST('TestPosUnderUpperBoundYes');
stPositionState.fPosition := 10;
stPositionState.fDelta := 1;

AssertTrue(
    Condition:=F_PosUnderUpperBound(
        fPosition:=10.9,
        stPositionState:=stPositionState,
    ),
    Message:='Decided 10.9 > 11.0',
);
TEST_FINISHED();
END_METHOD

METHOD PRIVATE TestPosWithinDeltaJustRight
VAR
    stPositionState: ST_PositionState;
END_VAR

TEST('TestPosWithinDeltaJustRight');
stPositionState.fPosition := 20;
stPositionState.fDelta := 1;

AssertTrue(
    Condition:=F_PosWithinDelta(
        fPosition:=20.2,
        stPositionState:=stPositionState,
    ),
    Message:='Decided 20.2 not within 19 to 21 bounds',
);
TEST_FINISHED();
END_METHOD

METHOD PRIVATE TestPosWithinDeltaTooHigh
VAR
    stPositionState: ST_PositionState;
END_VAR

TEST('TestPosWithinDeltaTooHigh');
stPositionState.fPosition := 20;
stPositionState.fDelta := 1;

AssertFalse(
    Condition:=F_PosWithinDelta(
        fPosition:=25.0,
        stPositionState:=stPositionState,
    ),
    Message:='Decided 21.0 > 25.0',
);
TEST_FINISHED();
END_METHOD

METHOD PRIVATE TestPosWithinDeltaTooLow
VAR
    stPositionState: ST_PositionState;
END_VAR

TEST('TestPosWithinDeltaTooLow');
stPositionState.fPosition := 20;
stPositionState.fDelta := 1;

AssertFalse(
    Condition:=F_PosWithinDelta(
        fPosition:=12.0,
        stPositionState:=stPositionState,
    ),
    Message:='Decided 12.0 > 19.0',
);
TEST_FINISHED();
END_METHOD

END_FUNCTION_BLOCK

// ---- POUs/Motion/FB_MotionStage.TcPOU
FUNCTION_BLOCK FB_MotionStage IMPLEMENTS I_MotionStage
(*
    Default implementation for PLC behavior when motor IOC asks for a move
    This can be extended or replaced in your PLC project if you want
    non-default behavior to arise from the motor record processing
*)
VAR_IN_OUT
    stMotionStage: ST_MotionStage;
END_VAR
VAR
    fbDriveVirtual: FB_DriveVirtual;
    fbMotionHome: FB_MotionHoming;
    fbSaveRestore: FB_EncSaveRestore;
    fbLogError: FB_LogMotionError;
    fbBacklashCompensation: FB_MotionBacklashCompensation;
    bExecute: BOOL;
    bExecMove: BOOL;
    bExecHome: BOOL;
    bFwdHit: BOOL;
    bBwdHit: BOOL;
    ftExec: F_TRIG;
    rtExec: R_TRIG;
    rtUserExec: R_TRIG;
    rtTarget: R_TRIG;
    rtHomed: R_TRIG;
    fbSetEnables: FB_SetEnables;
    bPosGoal: BOOL;
    bNegGoal: BOOL;
    fbEncoderValue: FB_EncoderValue;
    fbNCParams: FB_MotionStageNCParams;
    bNewMoveReq: BOOL;
    bPrepareDisable: BOOL;
    bMoveCmd: BOOL;
    rtMoveCmdShortcut: R_TRIG;
    rtHomeCmdShortcut: R_TRIG;
    rtEnableMode: R_TRIG;

    {attribute 'pytmc' := 'pv: '}
    stMotionStatus : ST_MotionStatus;
    stMotionCmdPrev : ST_MotionCommand;
    {attribute 'pytmc' := 'pv: '}
    stMotionCmdNow : ST_MotionCommand;
    {attribute 'pytmc' := 'pv: '}
    stExMotionStatus : ST_ExtendedMotionStatus;
    stMotionStageMethods : REFERENCE TO ST_MotionStage;
END_VAR


stMotionStageMethods REF= stMotionStage;

IF NOT __ISVALIDREF(stMotionStage) THEN
    RETURN;
END_IF

// Main Motion Command Structure
IF stMotionCmdNow.bHalt <> stMotionCmdPrev.bHalt THEN
    stMotionStage.bExecute := NOT stMotionCmdNow.bHalt;
END_IF
IF stMotionCmdNow.bHomeCmd <> stMotionCmdPrev.bHomeCmd THEN
    stMotionStage.bHomeCmd := stMotionCmdNow.bHomeCmd;
END_IF
IF stMotionCmdNow.bMoveCmd <> stMotionCmdPrev.bMoveCmd THEN
    stMotionStage.bMoveCmd := stMotionCmdNow.bMoveCmd;
END_IF
IF stMotionCmdNow.bReset <> stMotionCmdPrev.bReset THEN
    stMotionStage.bReset := stMotionCmdNow.bReset;
END_IF
IF stMotionCmdNow.fAcceleration <> stMotionCmdPrev.fAcceleration THEN
    stMotionStage.fAcceleration := stMotionCmdNow.fAcceleration;
END_IF
IF stMotionCmdNow.fDeceleration <> stMotionCmdPrev.fDeceleration THEN
    stMotionStage.fDeceleration := stMotionCmdNow.fDeceleration;
END_IF
IF stMotionCmdNow.fHomePosition <> stMotionCmdPrev.fHomePosition THEN
    stMotionStage.fHomePosition := stMotionCmdNow.fHomePosition;
END_IF
IF stMotionCmdNow.fJerk <> stMotionCmdPrev.fJerk THEN
    //stMotionStage.fJerk := stMotionCmdNow.fJerk; NOT SUPPORTED BY THIS IMPLEMENTATION
END_IF
IF stMotionCmdNow.fPosition <> stMotionCmdPrev.fPosition THEN
    stMotionStage.fPosition := stMotionCmdNow.fPosition;
END_IF
IF stMotionCmdNow.fVelocity <> stMotionCmdPrev.fVelocity THEN
    stMotionStage.fVelocity := stMotionCmdNow.fVelocity;
END_IF
IF stMotionCmdNow.nCmdData <> stMotionCmdPrev.nCmdData THEN
    stMotionStage.nCmdData := stMotionCmdNow.nCmdData;
END_IF
IF stMotionCmdNow.nCommand <> stMotionCmdPrev.nCommand THEN
    stMotionStage.nCommand := stMotionCmdNow.nCommand;
END_IF

// Start with an accurate status
stMotionStage.Axis.ReadStatus();

// Check for the plc shortcut commands
// Used for testing or to circumvent motor record issues
rtMoveCmdShortcut(CLK:=stMotionStage.bMoveCmd);
rtHomeCmdShortcut(CLK:=stMotionStage.bHomeCmd);
// Execute on rising edge
IF rtMoveCmdShortcut.Q AND NOT stMotionStage.bExecute THEN
    stMotionStage.bExecute := TRUE;
    stMotionStage.nCommand := E_EpicsMotorCmd.MOVE_ABSOLUTE;

    // attempting to move an axis without homing first?
    IF stMotionStage.nHomingMode <> E_EpicsHomeCmd.NONE AND NOT stMotionStage.bHomed THEN
        // one can just set bHome here even though no homing was done?
        stMotionStage.sErrorMessage := 'Axis homing mode set, but homing routine pending';
    END_IF

ELSIF rtHomeCmdShortcut.Q AND NOT stMotionStage.bExecute THEN
    stMotionStage.bExecute := TRUE;
    stMotionStage.nCommand := E_EpicsMotorCmd.HOME;
END_IF
// Always reset, even if not rising edge, so command can be issued again
IF stMotionStage.bMoveCmd OR stMotionStage.bHomeCmd THEN
    stMotionStage.bMoveCmd := FALSE;
    stMotionStage.bHomeCmd := FALSE;
END_IF

// Automatically fill the correct nCmdData for homing
IF stMotionStage.nCommand = E_EpicsMotorCmd.HOME THEN
    stMotionStage.nCmdData := stMotionStage.nHomingMode;
END_IF

// Check if the command wants to cause a move
bMoveCmd R= stMotionStage.nCmdData = E_EpicsHomeCmd.ABSOLUTE_SET;
bMoveCmd R= stMotionStage.nCmdData = E_EpicsHomeCmd.NONE;
bMoveCmd S= stMotionStage.nCommand <> E_EpicsMotorCmd.HOME;

// Handle main execs
rtUserExec(CLK := stMotionStage.bExecute);
bNewMoveReq S= rtUserExec.Q AND bMoveCmd;
bNewMoveReq R= NOT stMotionStage.bExecute;
bPrepareDisable R= bNewMoveReq;

bPosGoal := stMotionStage.stAxisStatus.fActPosition < stMotionStage.fPosition;
bNegGoal := stMotionStage.stAxisStatus.fActPosition > stMotionStage.fPosition;

// Moves are automatically allowed if no safety hooks. Otherwise, some other code will set this.
stMotionStage.bSafetyReady S= stMotionStage.bPowerSelf;

